LIN {X -76.668,Y -27.149,Z -45.520,A -90.000,B 90.000,C 0.000} C_DIS
LIN {X -76.579,Y -27.148,Z -45.468,A -90.000,B 90.000,C 0.000} C_DIS
LIN {X -76.520,Y -27.146,Z -45.437,A -90.000,B 90.000,C 0.000} C_DIS
LIN {X -76.472,Y -27.145,Z -45.413,A -90.000,B 90.000,C 0.000} C_DIS
LIN {X -76.330,Y -27.139,Z -45.352,A -90.000,B 90.000,C 0.000} C_DIS
LIN {X -76.220,Y -27.135,Z -45.309,A -90.000,B 90.000,C 0.000} C_DIS
LIN {X -75.832,Y -27.123,Z -45.175,A -90.000,B 90.000,C 0.000} C_DIS
LIN {X -75.654,Y -27.113,Z -45.115,A -90.000,B 90.000,C 0.000} C_DIS
LIN {X -75.440,Y -27.095,Z -45.043,A -90.000,B 90.000,C 0.000} C_DIS
LIN {X -75.320,Y -27.086,Z -45.007,A -90.000,B 90.000,C 0.000} C_DIS
LIN {X -75.000,Y -27.064,Z -44.932,A -90.000,B 90.000,C 0.000} C_DIS
LIN {X -74.933,Y -27.060,Z -44.917,A -90.000,B 90.000,C 0.000} C_DIS
LIN {X -74.743,Y -27.049,Z -44.886,A -90.000,B 90.000,C 0.000} C_DIS
LIN {X -74.638,Y -27.044,Z -44.876,A -90.000,B 90.000,C 0.000} C_DIS
LIN {X -74.553,Y -27.040,Z -44.872,A -90.000,B 90.000,C 0.000} C_DIS
LIN {X -74.405,Y -27.038,Z -44.874,A -90.000,B 90.000,C 0.000} C_DIS
LIN {X -74.238,Y -27.035,Z -44.881,A -90.000,B 90.000,C 0.000} C_DIS
LIN {X -74.171,Y -27.032,Z -44.885,A -90.000,B 90.000,C 0.000} C_DIS
LIN {X -74.041,Y -27.028,Z -44.899,A -90.000,B 90.000,C 0.000} C_DIS
LIN {X -73.894,Y -27.024,Z -44.925,A -90.000,B 90.000,C 0.000} C_DIS
LIN {X -73.078,Y -26.996,Z -45.023,A -90.000,B 90.000,C 0.000} C_DIS
LIN {X -72.681,Y -26.986,Z -45.070,A -90.000,B 90.000,C 0.000} C_DIS
LIN {X -72.606,Y -26.984,Z -45.081,A -90.000,B 90.000,C 0.000} C_DIS
LIN {X -72.312,Y -26.976,Z -45.155,A -90.000,B 90.000,C 0.000} C_DIS
LIN {X -72.076,Y -26.973,Z -45.234,A -90.000,B 90.000,C 0.000} C_DIS
LIN {X -72.048,Y -26.973,Z -45.245,A -90.000,B 90.000,C 0.000} C_DIS
LIN {X -71.550,Y -26.959,Z -45.362,A -90.000,B 90.000,C 0.000} C_DIS
LIN {X -71.035,Y -26.949,Z -45.481,A -90.000,B 90.000,C 0.000} C_DIS
LIN {X -70.942,Y -26.945,Z -45.503,A -90.000,B 90.000,C 0.000} C_DIS
LIN {X -70.816,Y -26.940,Z -45.537,A -90.000,B 90.000,C 0.000} C_DIS
LIN {X -70.607,Y -26.935,Z -45.607,A -90.000,B 90.000,C 0.000} C_DIS
LIN {X -70.486,Y -26.933,Z -45.651,A -90.000,B 90.000,C 0.000} C_DIS
LIN {X -69.761,Y -26.903,Z -45.823,A -90.000,B 90.000,C 0.000} C_DIS
LIN {X -69.366,Y -26.892,Z -45.916,A -90.000,B 90.000,C 0.000} C_DIS
LIN {X -69.227,Y -26.882,Z -45.922,A -90.000,B 90.000,C 0.000} C_DIS
LIN {X -69.048,Y -26.872,Z -45.944,A -90.000,B 90.000,C 0.000} C_DIS
LIN {X -68.707,Y -26.860,Z -46.014,A -90.000,B 90.000,C 0.000} C_DIS
LIN {X -67.594,Y -26.796,Z -46.253,A -90.000,B 90.000,C 0.000} C_DIS
LIN {X -67.151,Y -26.765,Z -46.342,A -90.000,B 90.000,C 0.000} C_DIS
LIN {X -66.963,Y -26.753,Z -46.384,A -90.000,B 90.000,C 0.000} C_DIS
LIN {X -66.920,Y -26.749,Z -46.390,A -90.000,B 90.000,C 0.000} C_DIS
LIN {X -66.399,Y -26.719,Z -46.458,A -90.000,B 90.000,C 0.000} C_DIS
LIN {X -66.250,Y -26.713,Z -46.485,A -90.000,B 90.000,C 0.000} C_DIS
LIN {X -66.013,Y -26.705,Z -46.537,A -90.000,B 90.000,C 0.000} C_DIS
LIN {X -65.089,Y -26.644,Z -46.751,A -90.000,B 90.000,C 0.000} C_DIS
LIN {X -64.621,Y -26.614,Z -46.860,A -90.000,B 90.000,C 0.000} C_DIS
LIN {X -64.516,Y -26.603,Z -46.873,A -90.000,B 90.000,C 0.000} C_DIS
LIN {X -64.385,Y -26.595,Z -46.892,A -90.000,B 90.000,C 0.000} C_DIS
LIN {X -64.154,Y -26.585,Z -46.933,A -90.000,B 90.000,C 0.000} C_DIS
LIN {X -63.476,Y -26.545,Z -47.056,A -90.000,B 90.000,C 0.000} C_DIS
LIN {X -63.310,Y -26.538,Z -47.093,A -90.000,B 90.000,C 0.000} C_DIS
LIN {X -63.159,Y -26.532,Z -47.128,A -90.000,B 90.000,C 0.000} C_DIS
LIN {X -61.858,Y -26.456,Z -47.450,A -90.000,B 90.000,C 0.000} C_DIS
LIN {X -61.801,Y -26.451,Z -47.460,A -90.000,B 90.000,C 0.000} C_DIS
LIN {X -61.487,Y -26.434,Z -47.509,A -90.000,B 90.000,C 0.000} C_DIS
LIN {X -61.371,Y -26.430,Z -47.531,A -90.000,B 90.000,C 0.000} C_DIS
LIN {X -61.170,Y -26.422,Z -47.574,A -90.000,B 90.000,C 0.000} C_DIS
LIN {X -60.377,Y -26.379,Z -47.754,A -90.000,B 90.000,C 0.000} C_DIS
LIN {X -59.277,Y -26.330,Z -48.032,A -90.000,B 90.000,C 0.000} C_DIS
LIN {X -59.103,Y -26.323,Z -48.077,A -90.000,B 90.000,C 0.000} C_DIS
LIN {X -59.005,Y -26.321,Z -48.100,A -90.000,B 90.000,C 0.000} C_DIS
LIN {X -58.397,Y -26.301,Z -48.215,A -90.000,B 90.000,C 0.000} C_DIS
LIN {X -58.186,Y -26.296,Z -48.262,A -90.000,B 90.000,C 0.000} C_DIS
LIN {X -57.425,Y -26.286,Z -48.443,A -90.000,B 90.000,C 0.000} C_DIS
LIN {X -56.485,Y -26.265,Z -48.675,A -90.000,B 90.000,C 0.000} C_DIS
LIN {X -55.979,Y -26.267,Z -48.792,A -90.000,B 90.000,C 0.000} C_DIS
LIN {X -55.691,Y -26.263,Z -48.851,A -90.000,B 90.000,C 0.000} C_DIS
LIN {X -54.901,Y -26.262,Z -49.008,A -90.000,B 90.000,C 0.000} C_DIS
LIN {X -54.076,Y -26.270,Z -49.199,A -90.000,B 90.000,C 0.000} C_DIS
LIN {X -52.954,Y -26.306,Z -49.443,A -90.000,B 90.000,C 0.000} C_DIS
LIN {X -51.548,Y -26.347,Z -49.740,A -90.000,B 90.000,C 0.000} C_DIS
LIN {X -51.220,Y -26.356,Z -49.809,A -90.000,B 90.000,C 0.000} C_DIS
LIN {X -50.961,Y -26.369,Z -49.862,A -90.000,B 90.000,C 0.000} C_DIS
LIN {X -50.773,Y -26.379,Z -49.904,A -90.000,B 90.000,C 0.000} C_DIS
LIN {X -50.032,Y -26.422,Z -50.072,A -90.000,B 90.000,C 0.000} C_DIS
LIN {X -49.104,Y -26.464,Z -50.267,A -90.000,B 90.000,C 0.000} C_DIS
LIN {X -48.814,Y -26.479,Z -50.333,A -90.000,B 90.000,C 0.000} C_DIS
LIN {X -48.233,Y -26.506,Z -50.468,A -90.000,B 90.000,C 0.000} C_DIS
LIN {X -47.893,Y -26.526,Z -50.543,A -90.000,B 90.000,C 0.000} C_DIS
LIN {X -47.412,Y -26.550,Z -50.637,A -90.000,B 90.000,C 0.000} C_DIS
LIN {X -46.971,Y -26.573,Z -50.730,A -90.000,B 90.000,C 0.000} C_DIS
LIN {X -46.694,Y -26.575,Z -50.762,A -90.000,B 90.000,C 0.000} C_DIS
LIN {X -45.976,Y -26.553,Z -50.795,A -90.000,B 90.000,C 0.000} C_DIS
LIN {X -45.116,Y -26.531,Z -50.839,A -90.000,B 90.000,C 0.000} C_DIS
LIN {X -44.321,Y -26.510,Z -50.871,A -90.000,B 90.000,C 0.000} C_DIS
LIN {X -43.871,Y -26.485,Z -50.896,A -90.000,B 90.000,C 0.000} C_DIS
LIN {X -42.715,Y -26.432,Z -50.983,A -90.000,B 90.000,C 0.000} C_DIS
LIN {X -42.367,Y -26.419,Z -51.020,A -90.000,B 90.000,C 0.000} C_DIS
LIN {X -41.622,Y -26.397,Z -51.105,A -90.000,B 90.000,C 0.000} C_DIS
LIN {X -40.921,Y -26.380,Z -51.187,A -90.000,B 90.000,C 0.000} C_DIS
LIN {X -39.390,Y -26.335,Z -51.371,A -90.000,B 90.000,C 0.000} C_DIS
LIN {X -39.171,Y -26.331,Z -51.405,A -90.000,B 90.000,C 0.000} C_DIS
LIN {X -38.129,Y -26.312,Z -51.576,A -90.000,B 90.000,C 0.000} C_DIS
LIN {X -37.797,Y -26.306,Z -51.632,A -90.000,B 90.000,C 0.000} C_DIS
LIN {X -37.029,Y -26.296,Z -51.768,A -90.000,B 90.000,C 0.000} C_DIS
LIN {X -36.278,Y -26.283,Z -51.903,A -90.000,B 90.000,C 0.000} C_DIS
LIN {X -35.844,Y -26.277,Z -51.985,A -90.000,B 90.000,C 0.000} C_DIS
LIN {X -35.325,Y -26.267,Z -52.085,A -90.000,B 90.000,C 0.000} C_DIS
LIN {X -33.082,Y -26.239,Z -52.548,A -90.000,B 90.000,C 0.000} C_DIS
LIN {X -32.307,Y -26.223,Z -52.710,A -90.000,B 90.000,C 0.000} C_DIS
LIN {X -31.608,Y -26.212,Z -52.862,A -90.000,B 90.000,C 0.000} C_DIS
LIN {X -30.365,Y -26.201,Z -53.148,A -90.000,B 90.000,C 0.000} C_DIS
LIN {X -29.820,Y -26.194,Z -53.275,A -90.000,B 90.000,C 0.000} C_DIS
LIN {X -29.558,Y -26.188,Z -53.337,A -90.000,B 90.000,C 0.000} C_DIS
LIN {X -29.212,Y -26.184,Z -53.417,A -90.000,B 90.000,C 0.000} C_DIS
LIN {X -27.279,Y -26.151,Z -53.851,A -90.000,B 90.000,C 0.000} C_DIS
LIN {X -26.462,Y -26.136,Z -54.036,A -90.000,B 90.000,C 0.000} C_DIS
LIN {X -26.354,Y -26.132,Z -54.059,A -90.000,B 90.000,C 0.000} C_DIS
LIN {X -24.983,Y -26.105,Z -54.333,A -90.000,B 90.000,C 0.000} C_DIS
LIN {X -24.301,Y -26.086,Z -54.456,A -90.000,B 90.000,C 0.000} C_DIS
LIN {X -23.848,Y -26.066,Z -54.528,A -90.000,B 90.000,C 0.000} C_DIS
LIN {X -23.603,Y -26.060,Z -54.564,A -90.000,B 90.000,C 0.000} C_DIS
LIN {X -23.357,Y -26.057,Z -54.597,A -90.000,B 90.000,C 0.000} C_DIS
LIN {X -22.651,Y -26.032,Z -54.669,A -90.000,B 90.000,C 0.000} C_DIS
LIN {X -22.402,Y -26.017,Z -54.685,A -90.000,B 90.000,C 0.000} C_DIS
LIN {X -22.145,Y -25.999,Z -54.688,A -90.000,B 90.000,C 0.000} C_DIS
LIN {X -21.779,Y -25.983,Z -54.683,A -90.000,B 90.000,C 0.000} C_DIS
LIN {X -21.198,Y -25.921,Z -54.631,A -90.000,B 90.000,C 0.000} C_DIS
LIN {X -21.158,Y -25.919,Z -54.625,A -90.000,B 90.000,C 0.000} C_DIS
LIN {X -20.482,Y -25.823,Z -54.462,A -90.000,B 90.000,C 0.000} C_DIS
LIN {X -20.459,Y -25.820,Z -54.457,A -90.000,B 90.000,C 0.000} C_DIS
LIN {X -20.316,Y -25.816,Z -54.414,A -90.000,B 90.000,C 0.000} C_DIS
LIN {X -19.976,Y -25.803,Z -54.320,A -90.000,B 90.000,C 0.000} C_DIS
LIN {X -19.491,Y -25.762,Z -54.163,A -90.000,B 90.000,C 0.000} C_DIS
LIN {X -19.170,Y -25.749,Z -54.042,A -90.000,B 90.000,C 0.000} C_DIS
LIN {X -18.511,Y -25.729,Z -53.805,A -90.000,B 90.000,C 0.000} C_DIS
LIN {X -18.354,Y -25.723,Z -53.745,A -90.000,B 90.000,C 0.000} C_DIS
LIN {X -17.302,Y -25.718,Z -53.351,A -90.000,B 90.000,C 0.000} C_DIS
LIN {X -16.990,Y -25.716,Z -53.234,A -90.000,B 90.000,C 0.000} C_DIS
LIN {X -16.551,Y -25.702,Z -53.087,A -90.000,B 90.000,C 0.000} C_DIS
LIN {X -16.275,Y -25.697,Z -52.992,A -90.000,B 90.000,C 0.000} C_DIS
LIN {X -15.804,Y -25.701,Z -52.842,A -90.000,B 90.000,C 0.000} C_DIS
LIN {X -15.519,Y -25.709,Z -52.757,A -90.000,B 90.000,C 0.000} C_DIS
LIN {X -14.893,Y -25.715,Z -52.585,A -90.000,B 90.000,C 0.000} C_DIS
LIN {X -14.842,Y -25.713,Z -52.574,A -90.000,B 90.000,C 0.000} C_DIS
LIN {X -14.139,Y -25.698,Z -52.428,A -90.000,B 90.000,C 0.000} C_DIS
LIN {X -13.133,Y -25.670,Z -52.234,A -90.000,B 90.000,C 0.000} C_DIS
LIN {X -12.867,Y -25.665,Z -52.190,A -90.000,B 90.000,C 0.000} C_DIS
LIN {X -12.574,Y -25.660,Z -52.144,A -90.000,B 90.000,C 0.000} C_DIS
LIN {X -11.885,Y -25.673,Z -52.058,A -90.000,B 90.000,C 0.000} C_DIS
LIN {X -11.634,Y -25.672,Z -52.037,A -90.000,B 90.000,C 0.000} C_DIS
LIN {X -11.198,Y -25.673,Z -52.007,A -90.000,B 90.000,C 0.000} C_DIS
LIN {X -10.131,Y -25.674,Z -51.968,A -90.000,B 90.000,C 0.000} C_DIS
LIN {X -9.127,Y -25.674,Z -51.924,A -90.000,B 90.000,C 0.000} C_DIS
LIN {X -9.054,Y -25.675,Z -51.922,A -90.000,B 90.000,C 0.000} C_DIS
LIN {X -8.312,Y -25.671,Z -51.917,A -90.000,B 90.000,C 0.000} C_DIS
LIN {X -7.938,Y -25.680,Z -51.922,A -90.000,B 90.000,C 0.000} C_DIS
LIN {X -7.084,Y -25.713,Z -51.944,A -90.000,B 90.000,C 0.000} C_DIS
LIN {X -6.515,Y -25.723,Z -51.975,A -90.000,B 90.000,C 0.000} C_DIS
LIN {X -5.811,Y -25.734,Z -52.016,A -90.000,B 90.000,C 0.000} C_DIS
LIN {X -5.328,Y -25.747,Z -52.047,A -90.000,B 90.000,C 0.000} C_DIS
LIN {X -4.775,Y -25.774,Z -52.093,A -90.000,B 90.000,C 0.000} C_DIS
LIN {X -3.453,Y -25.814,Z -52.238,A -90.000,B 90.000,C 0.000} C_DIS
LIN {X -2.718,Y -25.836,Z -52.319,A -90.000,B 90.000,C 0.000} C_DIS
LIN {X -2.230,Y -25.852,Z -52.374,A -90.000,B 90.000,C 0.000} C_DIS
LIN {X -1.872,Y -25.876,Z -52.429,A -90.000,B 90.000,C 0.000} C_DIS
LIN {X -0.557,Y -25.960,Z -52.642,A -90.000,B 90.000,C 0.000} C_DIS
LIN {X -0.166,Y -25.976,Z -52.698,A -90.000,B 90.000,C 0.000} C_DIS
LIN {X 0.552,Y -26.009,Z -52.808,A -90.000,B 90.000,C 0.000} C_DIS
LIN {X 0.727,Y -26.014,Z -52.838,A -90.000,B 90.000,C 0.000} C_DIS
LIN {X 0.921,Y -26.024,Z -52.878,A -90.000,B 90.000,C 0.000} C_DIS
LIN {X 1.351,Y -26.042,Z -52.975,A -90.000,B 90.000,C 0.000} C_DIS
LIN {X 1.495,Y -26.054,Z -53.002,A -90.000,B 90.000,C 0.000} C_DIS
LIN {X 2.799,Y -26.132,Z -53.211,A -90.000,B 90.000,C 0.000} C_DIS
LIN {X 3.009,Y -26.149,Z -53.251,A -90.000,B 90.000,C 0.000} C_DIS
LIN {X 3.118,Y -26.159,Z -53.272,A -90.000,B 90.000,C 0.000} C_DIS
LIN {X 3.768,Y -26.195,Z -53.373,A -90.000,B 90.000,C 0.000} C_DIS
LIN {X 4.343,Y -26.230,Z -53.460,A -90.000,B 90.000,C 0.000} C_DIS
LIN {X 4.515,Y -26.234,Z -53.477,A -90.000,B 90.000,C 0.000} C_DIS
LIN {X 4.986,Y -26.259,Z -53.514,A -90.000,B 90.000,C 0.000} C_DIS
LIN {X 5.416,Y -26.287,Z -53.555,A -90.000,B 90.000,C 0.000} C_DIS
LIN {X 5.715,Y -26.295,Z -53.563,A -90.000,B 90.000,C 0.000} C_DIS
LIN {X 6.310,Y -26.301,Z -53.557,A -90.000,B 90.000,C 0.000} C_DIS
LIN {X 6.763,Y -26.310,Z -53.550,A -90.000,B 90.000,C 0.000} C_DIS
LIN {X 7.708,Y -26.306,Z -53.477,A -90.000,B 90.000,C 0.000} C_DIS
LIN {X 8.237,Y -26.294,Z -53.427,A -90.000,B 90.000,C 0.000} C_DIS
LIN {X 8.504,Y -26.288,Z -53.400,A -90.000,B 90.000,C 0.000} C_DIS
LIN {X 9.112,Y -26.249,Z -53.356,A -90.000,B 90.000,C 0.000} C_DIS
LIN {X 9.378,Y -26.233,Z -53.345,A -90.000,B 90.000,C 0.000} C_DIS
LIN {X 9.815,Y -26.206,Z -53.332,A -90.000,B 90.000,C 0.000} C_DIS
LIN {X 9.935,Y -26.202,Z -53.332,A -90.000,B 90.000,C 0.000} C_DIS
LIN {X 10.931,Y -26.179,Z -53.355,A -90.000,B 90.000,C 0.000} C_DIS
LIN {X 11.248,Y -26.159,Z -53.373,A -90.000,B 90.000,C 0.000} C_DIS
LIN {X 11.681,Y -26.144,Z -53.417,A -90.000,B 90.000,C 0.000} C_DIS
LIN {X 11.767,Y -26.143,Z -53.430,A -90.000,B 90.000,C 0.000} C_DIS
LIN {X 12.047,Y -26.130,Z -53.483,A -90.000,B 90.000,C 0.000} C_DIS
LIN {X 12.477,Y -26.118,Z -53.558,A -90.000,B 90.000,C 0.000} C_DIS
LIN {X 12.961,Y -26.073,Z -53.618,A -90.000,B 90.000,C 0.000} C_DIS
LIN {X 13.125,Y -26.063,Z -53.643,A -90.000,B 90.000,C 0.000} C_DIS
LIN {X 13.751,Y -26.044,Z -53.760,A -90.000,B 90.000,C 0.000} C_DIS
LIN {X 14.266,Y -26.019,Z -53.825,A -90.000,B 90.000,C 0.000} C_DIS
LIN {X 14.500,Y -26.013,Z -53.861,A -90.000,B 90.000,C 0.000} C_DIS
LIN {X 14.939,Y -26.001,Z -53.932,A -90.000,B 90.000,C 0.000} C_DIS
LIN {X 15.047,Y -25.993,Z -53.945,A -90.000,B 90.000,C 0.000} C_DIS
LIN {X 15.382,Y -25.981,Z -53.980,A -90.000,B 90.000,C 0.000} C_DIS
LIN {X 15.560,Y -25.978,Z -54.003,A -90.000,B 90.000,C 0.000} C_DIS
LIN {X 15.976,Y -25.953,Z -54.039,A -90.000,B 90.000,C 0.000} C_DIS
LIN {X 16.371,Y -25.945,Z -54.086,A -90.000,B 90.000,C 0.000} C_DIS
LIN {X 16.524,Y -25.935,Z -54.097,A -90.000,B 90.000,C 0.000} C_DIS
LIN {X 16.741,Y -26.026,Z -54.021,A -90.000,B 90.000,C 0.000} C_DIS
LIN {X 16.808,Y -26.055,Z -54.000,A -90.000,B 90.000,C 0.000} C_DIS
LIN {X 16.933,Y -26.108,Z -53.971,A -90.000,B 90.000,C 0.000} C_DIS
LIN {X 17.083,Y -26.172,Z -53.944,A -90.000,B 90.000,C 0.000} C_DIS
LIN {X 17.196,Y -26.216,Z -53.927,A -90.000,B 90.000,C 0.000} C_DIS
LIN {X 17.303,Y -26.254,Z -53.911,A -90.000,B 90.000,C 0.000} C_DIS
LIN {X 17.592,Y -26.359,Z -53.877,A -90.000,B 90.000,C 0.000} C_DIS
LIN {X 17.749,Y -26.413,Z -53.864,A -90.000,B 90.000,C 0.000} C_DIS
LIN {X 17.828,Y -26.441,Z -53.862,A -90.000,B 90.000,C 0.000} C_DIS
LIN {X 18.139,Y -26.545,Z -53.863,A -90.000,B 90.000,C 0.000} C_DIS
LIN {X 18.300,Y -26.602,Z -53.870,A -90.000,B 90.000,C 0.000} C_DIS
LIN {X 18.401,Y -26.638,Z -53.867,A -90.000,B 90.000,C 0.000} C_DIS
LIN {X 18.613,Y -26.714,Z -53.875,A -90.000,B 90.000,C 0.000} C_DIS
LIN {X 18.655,Y -26.729,Z -53.880,A -90.000,B 90.000,C 0.000} C_DIS
LIN {X 18.754,Y -26.750,Z -53.795,A -90.000,B 90.000,C 0.000} C_DIS
LIN {X 18.774,Y -26.736,Z -53.643,A -90.000,B 90.000,C 0.000} C_DIS
LIN {X 18.828,Y -26.717,Z -53.412,A -90.000,B 90.000,C 0.000} C_DIS
LIN {X 18.955,Y -26.695,Z -53.020,A -90.000,B 90.000,C 0.000} C_DIS
LIN {X 19.026,Y -26.673,Z -52.812,A -90.000,B 90.000,C 0.000} C_DIS
LIN {X 19.080,Y -26.660,Z -52.672,A -90.000,B 90.000,C 0.000} C_DIS
LIN {X 19.259,Y -26.627,Z -52.252,A -90.000,B 90.000,C 0.000} C_DIS
LIN {X 19.331,Y -26.607,Z -52.091,A -90.000,B 90.000,C 0.000} C_DIS
LIN {X 19.446,Y -26.577,Z -51.845,A -90.000,B 90.000,C 0.000} C_DIS
LIN {X 19.492,Y -26.567,Z -51.753,A -90.000,B 90.000,C 0.000} C_DIS
LIN {X 19.554,Y -26.558,Z -51.644,A -90.000,B 90.000,C 0.000} C_DIS
LIN {X 19.612,Y -26.551,Z -51.554,A -90.000,B 90.000,C 0.000} C_DIS
LIN {X 19.696,Y -26.542,Z -51.430,A -90.000,B 90.000,C 0.000} C_DIS
LIN {X 19.880,Y -26.514,Z -51.172,A -90.000,B 90.000,C 0.000} C_DIS
LIN {X 20.028,Y -26.490,Z -50.967,A -90.000,B 90.000,C 0.000} C_DIS
LIN {X 20.210,Y -26.458,Z -50.712,A -90.000,B 90.000,C 0.000} C_DIS
LIN {X 20.290,Y -26.447,Z -50.610,A -90.000,B 90.000,C 0.000} C_DIS
LIN {X 20.384,Y -26.435,Z -50.495,A -90.000,B 90.000,C 0.000} C_DIS
LIN {X 20.492,Y -26.416,Z -50.351,A -90.000,B 90.000,C 0.000} C_DIS
LIN {X 20.559,Y -26.405,Z -50.264,A -90.000,B 90.000,C 0.000} C_DIS
LIN {X 20.692,Y -26.388,Z -50.109,A -90.000,B 90.000,C 0.000} C_DIS
LIN {X 20.911,Y -26.361,Z -49.879,A -90.000,B 90.000,C 0.000} C_DIS
LIN {X 21.128,Y -26.327,Z -49.657,A -90.000,B 90.000,C 0.000} C_DIS
LIN {X 21.369,Y -26.295,Z -49.419,A -90.000,B 90.000,C 0.000} C_DIS
LIN {X 21.491,Y -26.280,Z -49.298,A -90.000,B 90.000,C 0.000} C_DIS
LIN {X 21.593,Y -26.271,Z -49.204,A -90.000,B 90.000,C 0.000} C_DIS
LIN {X 21.776,Y -26.243,Z -49.013,A -90.000,B 90.000,C 0.000} C_DIS
LIN {X 21.928,Y -26.228,Z -48.873,A -90.000,B 90.000,C 0.000} C_DIS
LIN {X 22.146,Y -26.201,Z -48.678,A -90.000,B 90.000,C 0.000} C_DIS
LIN {X 22.398,Y -26.169,Z -48.453,A -90.000,B 90.000,C 0.000} C_DIS
LIN {X 22.719,Y -26.122,Z -48.184,A -90.000,B 90.000,C 0.000} C_DIS
LIN {X 22.870,Y -26.096,Z -48.043,A -90.000,B 90.000,C 0.000} C_DIS
LIN {X 23.304,Y -26.044,Z -47.683,A -90.000,B 90.000,C 0.000} C_DIS
LIN {X 23.430,Y -26.028,Z -47.580,A -90.000,B 90.000,C 0.000} C_DIS
LIN {X 23.577,Y -26.006,Z -47.467,A -90.000,B 90.000,C 0.000} C_DIS
LIN {X 23.702,Y -25.988,Z -47.374,A -90.000,B 90.000,C 0.000} C_DIS
LIN {X 23.939,Y -25.949,Z -47.209,A -90.000,B 90.000,C 0.000} C_DIS
LIN {X 23.988,Y -25.939,Z -47.172,A -90.000,B 90.000,C 0.000} C_DIS
LIN {X 24.179,Y -25.908,Z -47.041,A -90.000,B 90.000,C 0.000} C_DIS
LIN {X 24.532,Y -25.864,Z -46.789,A -90.000,B 90.000,C 0.000} C_DIS
LIN {X 24.820,Y -25.823,Z -46.595,A -90.000,B 90.000,C 0.000} C_DIS
LIN {X 25.032,Y -25.794,Z -46.461,A -90.000,B 90.000,C 0.000} C_DIS
LIN {X 25.512,Y -25.738,Z -46.177,A -90.000,B 90.000,C 0.000} C_DIS
LIN {X 25.704,Y -25.713,Z -46.074,A -90.000,B 90.000,C 0.000} C_DIS
LIN {X 25.770,Y -25.706,Z -46.039,A -90.000,B 90.000,C 0.000} C_DIS
LIN {X 25.938,Y -25.679,Z -45.945,A -90.000,B 90.000,C 0.000} C_DIS
LIN {X 25.999,Y -25.672,Z -45.913,A -90.000,B 90.000,C 0.000} C_DIS
LIN {X 26.061,Y -25.662,Z -45.884,A -90.000,B 90.000,C 0.000} C_DIS
LIN {X 26.279,Y -25.639,Z -45.764,A -90.000,B 90.000,C 0.000} C_DIS
LIN {X 26.350,Y -25.630,Z -45.729,A -90.000,B 90.000,C 0.000} C_DIS
LIN {X 26.679,Y -25.600,Z -45.574,A -90.000,B 90.000,C 0.000} C_DIS
LIN {X 26.829,Y -25.586,Z -45.504,A -90.000,B 90.000,C 0.000} C_DIS
LIN {X 27.144,Y -25.554,Z -45.370,A -90.000,B 90.000,C 0.000} C_DIS
LIN {X 27.283,Y -25.545,Z -45.313,A -90.000,B 90.000,C 0.000} C_DIS
LIN {X 27.612,Y -25.519,Z -45.199,A -90.000,B 90.000,C 0.000} C_DIS
LIN {X 27.822,Y -25.503,Z -45.125,A -90.000,B 90.000,C 0.000} C_DIS
LIN {X 28.017,Y -25.494,Z -45.048,A -90.000,B 90.000,C 0.000} C_DIS
LIN {X 28.430,Y -25.472,Z -44.901,A -90.000,B 90.000,C 0.000} C_DIS
LIN {X 28.884,Y -25.440,Z -44.766,A -90.000,B 90.000,C 0.000} C_DIS
LIN {X 29.328,Y -25.418,Z -44.640,A -90.000,B 90.000,C 0.000} C_DIS
LIN {X 29.665,Y -25.409,Z -44.546,A -90.000,B 90.000,C 0.000} C_DIS
LIN {X 30.143,Y -25.387,Z -44.458,A -90.000,B 90.000,C 0.000} C_DIS
LIN {X 30.385,Y -25.381,Z -44.414,A -90.000,B 90.000,C 0.000} C_DIS
LIN {X 30.701,Y -25.375,Z -44.351,A -90.000,B 90.000,C 0.000} C_DIS
LIN {X 30.921,Y -25.375,Z -44.308,A -90.000,B 90.000,C 0.000} C_DIS
LIN {X 31.396,Y -25.369,Z -44.241,A -90.000,B 90.000,C 0.000} C_DIS
LIN {X 31.533,Y -25.366,Z -44.225,A -90.000,B 90.000,C 0.000} C_DIS
LIN {X 31.992,Y -25.366,Z -44.150,A -90.000,B 90.000,C 0.000} C_DIS
LIN {X 32.576,Y -25.362,Z -44.091,A -90.000,B 90.000,C 0.000} C_DIS
LIN {X 32.639,Y -25.362,Z -44.084,A -90.000,B 90.000,C 0.000} C_DIS
LIN {X 33.254,Y -25.365,Z -44.001,A -90.000,B 90.000,C 0.000} C_DIS
LIN {X 33.639,Y -25.384,Z -43.913,A -90.000,B 90.000,C 0.000} C_DIS
LIN {X 34.121,Y -25.420,Z -43.779,A -90.000,B 90.000,C 0.000} C_DIS
LIN {X 34.426,Y -25.447,Z -43.697,A -90.000,B 90.000,C 0.000} C_DIS
LIN {X 34.840,Y -25.491,Z -43.589,A -90.000,B 90.000,C 0.000} C_DIS
LIN {X 35.180,Y -25.532,Z -43.503,A -90.000,B 90.000,C 0.000} C_DIS
LIN {X 35.643,Y -25.595,Z -43.382,A -90.000,B 90.000,C 0.000} C_DIS
LIN {X 35.904,Y -25.637,Z -43.319,A -90.000,B 90.000,C 0.000} C_DIS
LIN {X 36.220,Y -25.677,Z -43.233,A -90.000,B 90.000,C 0.000} C_DIS
LIN {X 36.547,Y -25.697,Z -43.128,A -90.000,B 90.000,C 0.000} C_DIS
LIN {X 37.209,Y -25.708,Z -42.887,A -90.000,B 90.000,C 0.000} C_DIS
LIN {X 37.591,Y -25.709,Z -42.757,A -90.000,B 90.000,C 0.000} C_DIS
LIN {X 38.265,Y -25.703,Z -42.524,A -90.000,B 90.000,C 0.000} C_DIS
LIN {X 39.037,Y -25.689,Z -42.263,A -90.000,B 90.000,C 0.000} C_DIS
LIN {X 39.260,Y -25.683,Z -42.190,A -90.000,B 90.000,C 0.000} C_DIS
LIN {X 39.448,Y -25.682,Z -42.131,A -90.000,B 90.000,C 0.000} C_DIS
LIN {X 40.472,Y -25.649,Z -41.869,A -90.000,B 90.000,C 0.000} C_DIS
LIN {X 40.807,Y -25.638,Z -41.786,A -90.000,B 90.000,C 0.000} C_DIS
LIN {X 40.945,Y -25.635,Z -41.753,A -90.000,B 90.000,C 0.000} C_DIS
LIN {X 41.621,Y -25.601,Z -41.626,A -90.000,B 90.000,C 0.000} C_DIS
LIN {X 42.277,Y -25.590,Z -41.517,A -90.000,B 90.000,C 0.000} C_DIS
LIN {X 42.441,Y -25.586,Z -41.493,A -90.000,B 90.000,C 0.000} C_DIS
LIN {X 42.768,Y -25.584,Z -41.450,A -90.000,B 90.000,C 0.000} C_DIS
LIN {X 42.836,Y -25.581,Z -41.444,A -90.000,B 90.000,C 0.000} C_DIS
LIN {X 43.470,Y -25.549,Z -41.413,A -90.000,B 90.000,C 0.000} C_DIS
LIN {X 43.740,Y -25.536,Z -41.407,A -90.000,B 90.000,C 0.000} C_DIS
LIN {X 44.495,Y -25.521,Z -41.402,A -90.000,B 90.000,C 0.000} C_DIS
LIN {X 44.954,Y -25.510,Z -41.405,A -90.000,B 90.000,C 0.000} C_DIS
LIN {X 45.185,Y -25.496,Z -41.424,A -90.000,B 90.000,C 0.000} C_DIS
LIN {X 45.672,Y -25.474,Z -41.464,A -90.000,B 90.000,C 0.000} C_DIS
LIN {X 45.840,Y -25.472,Z -41.480,A -90.000,B 90.000,C 0.000} C_DIS
LIN {X 46.338,Y -25.470,Z -41.531,A -90.000,B 90.000,C 0.000} C_DIS
LIN {X 46.541,Y -25.470,Z -41.554,A -90.000,B 90.000,C 0.000} C_DIS
LIN {X 46.945,Y -25.470,Z -41.607,A -90.000,B 90.000,C 0.000} C_DIS
LIN {X 46.969,Y -25.470,Z -41.610,A -90.000,B 90.000,C 0.000} C_DIS
LIN {X 47.006,Y -25.470,Z -41.616,A -90.000,B 90.000,C 0.000} C_DIS
LIN {X 47.631,Y -25.452,Z -41.759,A -90.000,B 90.000,C 0.000} C_DIS
LIN {X 48.069,Y -25.437,Z -41.870,A -90.000,B 90.000,C 0.000} C_DIS
LIN {X 49.214,Y -25.419,Z -42.200,A -90.000,B 90.000,C 0.000} C_DIS
LIN {X 49.936,Y -25.396,Z -42.449,A -90.000,B 90.000,C 0.000} C_DIS
LIN {X 50.448,Y -25.395,Z -42.631,A -90.000,B 90.000,C 0.000} C_DIS
LIN {X 50.890,Y -25.395,Z -42.799,A -90.000,B 90.000,C 0.000} C_DIS
LIN {X 51.270,Y -25.390,Z -42.968,A -90.000,B 90.000,C 0.000} C_DIS
LIN {X 51.726,Y -25.382,Z -43.186,A -90.000,B 90.000,C 0.000} C_DIS
LIN {X 52.514,Y -25.375,Z -43.567,A -90.000,B 90.000,C 0.000} C_DIS
LIN {X 52.832,Y -25.375,Z -43.721,A -90.000,B 90.000,C 0.000} C_DIS
LIN {X 53.252,Y -25.371,Z -43.942,A -90.000,B 90.000,C 0.000} C_DIS
LIN {X 53.731,Y -25.369,Z -44.197,A -90.000,B 90.000,C 0.000} C_DIS
LIN {X 54.062,Y -25.373,Z -44.381,A -90.000,B 90.000,C 0.000} C_DIS
LIN {X 54.663,Y -25.366,Z -44.782,A -90.000,B 90.000,C 0.000} C_DIS
LIN {X 55.983,Y -25.353,Z -45.672,A -90.000,B 90.000,C 0.000} C_DIS
LIN {X 56.709,Y -25.348,Z -46.165,A -90.000,B 90.000,C 0.000} C_DIS
LIN {X 56.970,Y -25.353,Z -46.344,A -90.000,B 90.000,C 0.000} C_DIS
LIN {X 57.628,Y -25.350,Z -46.890,A -90.000,B 90.000,C 0.000} C_DIS
LIN {X 58.716,Y -25.347,Z -47.797,A -90.000,B 90.000,C 0.000} C_DIS
LIN {X 59.365,Y -25.346,Z -48.341,A -90.000,B 90.000,C 0.000} C_DIS
LIN {X 59.550,Y -25.348,Z -48.500,A -90.000,B 90.000,C 0.000} C_DIS
LIN {X 61.659,Y -25.345,Z -50.511,A -90.000,B 90.000,C 0.000} C_DIS
LIN {X 62.243,Y -25.345,Z -51.065,A -90.000,B 90.000,C 0.000} C_DIS
LIN {X 63.430,Y -25.345,Z -52.210,A -90.000,B 90.000,C 0.000} C_DIS
LIN {X 64.546,Y -25.350,Z -53.168,A -90.000,B 90.000,C 0.000} C_DIS
LIN {X 65.143,Y -25.352,Z -53.696,A -90.000,B 90.000,C 0.000} C_DIS
LIN {X 65.281,Y -25.355,Z -53.797,A -90.000,B 90.000,C 0.000} C_DIS
LIN {X 65.888,Y -25.358,Z -54.242,A -90.000,B 90.000,C 0.000} C_DIS
LIN {X 66.397,Y -25.363,Z -54.599,A -90.000,B 90.000,C 0.000} C_DIS
LIN {X 67.106,Y -25.368,Z -55.095,A -90.000,B 90.000,C 0.000} C_DIS
LIN {X 67.414,Y -25.371,Z -55.299,A -90.000,B 90.000,C 0.000} C_DIS
LIN {X 68.034,Y -25.378,Z -55.694,A -90.000,B 90.000,C 0.000} C_DIS
LIN {X 68.809,Y -25.383,Z -56.188,A -90.000,B 90.000,C 0.000} C_DIS
LIN {X 69.269,Y -25.385,Z -56.487,A -90.000,B 90.000,C 0.000} C_DIS
LIN {X 70.843,Y -25.406,Z -57.499,A -90.000,B 90.000,C 0.000} C_DIS
LIN {X 71.243,Y -25.409,Z -57.758,A -90.000,B 90.000,C 0.000} C_DIS
LIN {X 71.440,Y -25.406,Z -57.903,A -90.000,B 90.000,C 0.000} C_DIS
LIN {X 71.833,Y -25.411,Z -58.194,A -90.000,B 90.000,C 0.000} C_DIS
LIN {X 73.108,Y -25.432,Z -59.117,A -90.000,B 90.000,C 0.000} C_DIS
LIN {X 73.479,Y -25.429,Z -59.415,A -90.000,B 90.000,C 0.000} C_DIS
LIN {X 73.640,Y -25.426,Z -59.560,A -90.000,B 90.000,C 0.000} C_DIS
LIN {X 74.219,Y -25.434,Z -60.092,A -90.000,B 90.000,C 0.000} C_DIS
LIN {X 74.389,Y -25.435,Z -60.255,A -90.000,B 90.000,C 0.000} C_DIS
LIN {X 75.003,Y -25.443,Z -60.849,A -90.000,B 90.000,C 0.000} C_DIS
LIN {X 75.340,Y -25.445,Z -61.186,A -90.000,B 90.000,C 0.000} C_DIS
LIN {X 75.477,Y -25.442,Z -61.339,A -90.000,B 90.000,C 0.000} C_DIS
LIN {X 75.641,Y -25.444,Z -61.526,A -90.000,B 90.000,C 0.000} C_DIS
LIN {X 75.828,Y -25.445,Z -61.749,A -90.000,B 90.000,C 0.000} C_DIS
LIN {X 76.797,Y -25.464,Z -62.921,A -90.000,B 90.000,C 0.000} C_DIS
LIN {X 77.048,Y -25.462,Z -63.259,A -90.000,B 90.000,C 0.000} C_DIS
LIN {X 77.113,Y -25.464,Z -63.349,A -90.000,B 90.000,C 0.000} C_DIS
LIN {X 77.827,Y -25.475,Z -64.382,A -90.000,B 90.000,C 0.000} C_DIS
LIN {X 78.100,Y -25.474,Z -64.792,A -90.000,B 90.000,C 0.000} C_DIS
LIN {X 78.318,Y -25.377,Z -65.060,A -90.000,B 90.000,C 0.000} C_DIS
LIN {X 78.477,Y -25.332,Z -65.279,A -90.000,B 90.000,C 0.000} C_DIS
LIN {X 78.538,Y -25.321,Z -65.365,A -90.000,B 90.000,C 0.000} C_DIS
LIN {X 79.023,Y -25.318,Z -63.714,A -90.000,B 90.000,C 0.000} C_DIS
LIN {X 79.744,Y -25.318,Z -61.550,A -90.000,B 90.000,C 0.000} C_DIS
LIN {X 79.787,Y -25.318,Z -61.437,A -90.000,B 90.000,C 0.000} C_DIS
LIN {X 80.297,Y -25.329,Z -59.799,A -90.000,B 90.000,C 0.000} C_DIS
LIN {X 80.458,Y -25.332,Z -59.321,A -90.000,B 90.000,C 0.000} C_DIS
LIN {X 80.594,Y -25.335,Z -58.952,A -90.000,B 90.000,C 0.000} C_DIS
LIN {X 81.205,Y -25.331,Z -57.294,A -90.000,B 90.000,C 0.000} C_DIS
LIN {X 81.757,Y -25.327,Z -56.054,A -90.000,B 90.000,C 0.000} C_DIS
LIN {X 82.142,Y -25.329,Z -55.094,A -90.000,B 90.000,C 0.000} C_DIS
LIN {X 82.335,Y -25.332,Z -54.668,A -90.000,B 90.000,C 0.000} C_DIS
LIN {X 83.333,Y -25.328,Z -52.807,A -90.000,B 90.000,C 0.000} C_DIS
LIN {X 83.588,Y -25.329,Z -52.374,A -90.000,B 90.000,C 0.000} C_DIS
LIN {X 84.750,Y -25.320,Z -50.668,A -90.000,B 90.000,C 0.000} C_DIS
LIN {X 85.030,Y -25.320,Z -50.285,A -90.000,B 90.000,C 0.000} C_DIS
LIN {X 86.348,Y -25.311,Z -48.702,A -90.000,B 90.000,C 0.000} C_DIS
LIN {X 86.674,Y -25.311,Z -48.342,A -90.000,B 90.000,C 0.000} C_DIS
LIN {X 88.117,Y -25.309,Z -46.880,A -90.000,B 90.000,C 0.000} C_DIS
LIN {X 88.495,Y -25.309,Z -46.539,A -90.000,B 90.000,C 0.000} C_DIS
LIN {X 89.960,Y -25.320,Z -45.253,A -90.000,B 90.000,C 0.000} C_DIS
LIN {X 90.061,Y -25.308,Z -45.164,A -90.000,B 90.000,C 0.000} C_DIS
LIN {X 90.061,Y -60.000,Z -45.164,A -90.000,B 90.000,C 0.000} C_DIS
LIN {X 116.506,Y -60.000,Z -47.954,A -90.000,B 90.000,C 0.000} C_DIS
LIN {X 116.506,Y -25.308,Z -47.954,A -90.000,B 90.000,C 0.000} C_DIS
LIN {X 116.372,Y -25.308,Z -48.278,A -90.000,B 90.000,C 0.000} C_DIS
LIN {X 116.294,Y -25.308,Z -48.466,A -90.000,B 90.000,C 0.000} C_DIS
LIN {X 116.211,Y -25.308,Z -48.654,A -90.000,B 90.000,C 0.000} C_DIS
LIN {X 116.177,Y -25.308,Z -48.721,A -90.000,B 90.000,C 0.000} C_DIS
LIN {X 116.166,Y -25.308,Z -48.738,A -90.000,B 90.000,C 0.000} C_DIS
LIN {X 116.156,Y -25.308,Z -48.745,A -90.000,B 90.000,C 0.000} C_DIS
LIN {X 116.162,Y -25.308,Z -48.741,A -90.000,B 90.000,C 0.000} C_DIS
LIN {X 116.162,Y -25.307,Z -48.731,A -90.000,B 90.000,C 0.000} C_DIS
LIN {X 116.173,Y -25.308,Z -48.707,A -90.000,B 90.000,C 0.000} C_DIS
LIN {X 116.173,Y -35.308,Z -48.706,A -90.000,B 90.000,C 0.000} C_DIS
LIN {X 116.175,Y -35.622,Z -48.699,A -90.000,B 90.000,C 0.000} C_DIS
LIN {X 116.178,Y -35.718,Z -48.683,A -90.000,B 90.000,C 0.000} C_DIS
LIN {X 116.188,Y -35.846,Z -48.646,A -90.000,B 90.000,C 0.000} C_DIS
LIN {X 116.216,Y -36.039,Z -48.549,A -90.000,B 90.000,C 0.000} C_DIS
LIN {X 116.254,Y -36.204,Z -48.425,A -90.000,B 90.000,C 0.000} C_DIS
LIN {X 116.301,Y -36.351,Z -48.277,A -90.000,B 90.000,C 0.000} C_DIS
LIN {X 116.356,Y -36.460,Z -48.108,A -90.000,B 90.000,C 0.000} C_DIS
LIN {X 116.418,Y -36.546,Z -47.923,A -90.000,B 90.000,C 0.000} C_DIS
LIN {X 116.558,Y -36.717,Z -47.516,A -90.000,B 90.000,C 0.000} C_DIS
LIN {X 116.710,Y -36.871,Z -47.082,A -90.000,B 90.000,C 0.000} C_DIS
LIN {X 116.787,Y -36.886,Z -46.863,A -90.000,B 90.000,C 0.000} C_DIS
LIN {X 116.864,Y -36.874,Z -46.649,A -90.000,B 90.000,C 0.000} C_DIS
LIN {X 117.012,Y -36.837,Z -46.244,A -90.000,B 90.000,C 0.000} C_DIS
LIN {X 117.080,Y -36.806,Z -46.061,A -90.000,B 90.000,C 0.000} C_DIS
LIN {X 117.143,Y -36.735,Z -45.896,A -90.000,B 90.000,C 0.000} C_DIS
LIN {X 117.200,Y -36.633,Z -45.751,A -90.000,B 90.000,C 0.000} C_DIS
LIN {X 117.248,Y -36.508,Z -45.630,A -90.000,B 90.000,C 0.000} C_DIS
LIN {X 117.288,Y -36.352,Z -45.537,A -90.000,B 90.000,C 0.000} C_DIS
LIN {X 117.304,Y -36.250,Z -45.503,A -90.000,B 90.000,C 0.000} C_DIS
LIN {X 117.317,Y -36.098,Z -45.476,A -90.000,B 90.000,C 0.000} C_DIS
LIN {X 117.320,Y -36.031,Z -45.471,A -90.000,B 90.000,C 0.000} C_DIS
LIN {X 117.321,Y -25.306,Z -45.468,A -90.000,B 90.000,C 0.000} C_DIS
LIN {X 117.327,Y -25.308,Z -45.447,A -90.000,B 90.000,C 0.000} C_DIS
LIN {X 117.325,Y -25.307,Z -45.451,A -90.000,B 90.000,C 0.000} C_DIS
LIN {X 117.328,Y -25.308,Z -45.442,A -90.000,B 90.000,C 0.000} C_DIS
LIN {X 117.326,Y -25.308,Z -45.472,A -90.000,B 90.000,C 0.000} C_DIS
LIN {X 117.320,Y -25.308,Z -45.504,A -90.000,B 90.000,C 0.000} C_DIS
LIN {X 117.264,Y -25.306,Z -45.746,A -90.000,B 90.000,C 0.000} C_DIS
LIN {X 117.200,Y -25.308,Z -45.940,A -90.000,B 90.000,C 0.000} C_DIS
LIN {X 117.121,Y -25.308,Z -46.207,A -90.000,B 90.000,C 0.000} C_DIS
LIN {X 117.121,Y -60.000,Z -46.207,A -90.000,B 90.000,C 0.000} C_DIS
LIN {X 101.846,Y -60.000,Z -82.605,A -90.000,B 90.000,C 0.000} C_DIS
LIN {X 101.846,Y -25.308,Z -82.605,A -90.000,B 90.000,C 0.000} C_DIS
LIN {X 101.717,Y -25.322,Z -82.799,A -90.000,B 90.000,C 0.000} C_DIS
LIN {X 101.429,Y -25.308,Z -83.230,A -90.000,B 90.000,C 0.000} C_DIS
LIN {X 101.429,Y -60.000,Z -83.230,A -90.000,B 90.000,C 0.000} C_DIS
LIN {X 16.086,Y -60.000,Z -52.149,A -90.000,B 90.000,C 0.000} C_DIS
LIN {X 16.086,Y -25.308,Z -52.149,A -90.000,B 90.000,C 0.000} C_DIS
LIN {X 16.213,Y -25.363,Z -52.142,A -90.000,B 90.000,C 0.000} C_DIS
LIN {X 16.390,Y -25.443,Z -52.140,A -90.000,B 90.000,C 0.000} C_DIS
LIN {X 16.520,Y -25.490,Z -52.103,A -90.000,B 90.000,C 0.000} C_DIS
LIN {X 16.722,Y -25.566,Z -52.058,A -90.000,B 90.000,C 0.000} C_DIS
LIN {X 16.952,Y -25.656,Z -52.016,A -90.000,B 90.000,C 0.000} C_DIS
LIN {X 17.252,Y -25.773,Z -51.970,A -90.000,B 90.000,C 0.000} C_DIS
LIN {X 17.406,Y -25.835,Z -51.951,A -90.000,B 90.000,C 0.000} C_DIS
LIN {X 17.445,Y -25.823,Z -51.866,A -90.000,B 90.000,C 0.000} C_DIS
LIN {X 17.549,Y -25.787,Z -51.645,A -90.000,B 90.000,C 0.000} C_DIS
LIN {X 17.636,Y -25.754,Z -51.461,A -90.000,B 90.000,C 0.000} C_DIS
LIN {X 17.804,Y -25.691,Z -51.126,A -90.000,B 90.000,C 0.000} C_DIS
LIN {X 17.860,Y -25.671,Z -51.024,A -90.000,B 90.000,C 0.000} C_DIS
LIN {X 17.926,Y -25.651,Z -50.912,A -90.000,B 90.000,C 0.000} C_DIS
LIN {X 17.989,Y -25.633,Z -50.809,A -90.000,B 90.000,C 0.000} C_DIS
LIN {X 18.097,Y -25.610,Z -50.649,A -90.000,B 90.000,C 0.000} C_DIS
LIN {X 18.237,Y -25.584,Z -50.452,A -90.000,B 90.000,C 0.000} C_DIS
LIN {X 18.309,Y -25.570,Z -50.355,A -90.000,B 90.000,C 0.000} C_DIS
LIN {X 18.578,Y -25.505,Z -50.002,A -90.000,B 90.000,C 0.000} C_DIS
LIN {X 18.760,Y -25.452,Z -49.771,A -90.000,B 90.000,C 0.000} C_DIS
LIN {X 18.887,Y -25.420,Z -49.621,A -90.000,B 90.000,C 0.000} C_DIS
LIN {X 18.977,Y -25.403,Z -49.516,A -90.000,B 90.000,C 0.000} C_DIS
LIN {X 19.136,Y -25.364,Z -49.321,A -90.000,B 90.000,C 0.000} C_DIS
LIN {X 19.242,Y -25.339,Z -49.201,A -90.000,B 90.000,C 0.000} C_DIS
LIN {X 19.394,Y -25.308,Z -49.037,A -90.000,B 90.000,C 0.000} C_DIS
LIN {X 19.394,Y -60.000,Z -49.037,A -90.000,B 90.000,C 0.000} C_DIS
LIN {X -88.319,Y -60.000,Z -44.460,A -90.000,B 90.000,C 0.000} C_DIS
LIN {X -88.319,Y -25.308,Z -44.460,A -90.000,B 90.000,C 0.000} C_DIS
LIN {X -88.092,Y -25.358,Z -44.495,A -90.000,B 90.000,C 0.000} C_DIS
LIN {X -87.820,Y -25.417,Z -44.541,A -90.000,B 90.000,C 0.000} C_DIS
LIN {X -87.508,Y -25.486,Z -44.598,A -90.000,B 90.000,C 0.000} C_DIS
LIN {X -87.286,Y -25.534,Z -44.648,A -90.000,B 90.000,C 0.000} C_DIS
LIN {X -86.917,Y -25.610,Z -44.752,A -90.000,B 90.000,C 0.000} C_DIS
LIN {X -86.738,Y -25.647,Z -44.809,A -90.000,B 90.000,C 0.000} C_DIS
LIN {X -86.219,Y -25.753,Z -44.985,A -90.000,B 90.000,C 0.000} C_DIS
LIN {X -85.906,Y -25.817,Z -45.101,A -90.000,B 90.000,C 0.000} C_DIS
LIN {X -85.568,Y -25.885,Z -45.232,A -90.000,B 90.000,C 0.000} C_DIS
LIN {X -85.146,Y -25.969,Z -45.407,A -90.000,B 90.000,C 0.000} C_DIS
LIN {X -84.809,Y -26.033,Z -45.556,A -90.000,B 90.000,C 0.000} C_DIS
LIN {X -84.397,Y -26.106,Z -45.743,A -90.000,B 90.000,C 0.000} C_DIS
LIN {X -84.316,Y -26.120,Z -45.781,A -90.000,B 90.000,C 0.000} C_DIS
LIN {X -84.120,Y -26.158,Z -45.829,A -90.000,B 90.000,C 0.000} C_DIS
LIN {X -83.827,Y -26.214,Z -45.904,A -90.000,B 90.000,C 0.000} C_DIS
LIN {X -83.684,Y -26.240,Z -45.946,A -90.000,B 90.000,C 0.000} C_DIS
LIN {X -83.538,Y -26.267,Z -45.993,A -90.000,B 90.000,C 0.000} C_DIS
LIN {X -83.010,Y -26.364,Z -46.171,A -90.000,B 90.000,C 0.000} C_DIS
LIN {X -82.652,Y -26.418,Z -46.290,A -90.000,B 90.000,C 0.000} C_DIS
LIN {X -82.393,Y -26.457,Z -46.383,A -90.000,B 90.000,C 0.000} C_DIS
LIN {X -81.680,Y -26.573,Z -46.648,A -90.000,B 90.000,C 0.000} C_DIS
LIN {X -81.388,Y -26.620,Z -46.762,A -90.000,B 90.000,C 0.000} C_DIS
LIN {X -81.205,Y -26.649,Z -46.840,A -90.000,B 90.000,C 0.000} C_DIS
LIN {X -80.886,Y -26.694,Z -46.994,A -90.000,B 90.000,C 0.000} C_DIS
LIN {X -80.329,Y -26.763,Z -47.264,A -90.000,B 90.000,C 0.000} C_DIS
LIN {X -80.024,Y -26.800,Z -47.418,A -90.000,B 90.000,C 0.000} C_DIS
LIN {X -79.687,Y -26.842,Z -47.584,A -90.000,B 90.000,C 0.000} C_DIS
LIN {X -79.656,Y -26.865,Z -47.387,A -90.000,B 90.000,C 0.000} C_DIS
LIN {X -79.647,Y -26.870,Z -47.343,A -90.000,B 90.000,C 0.000} C_DIS
LIN {X -79.640,Y -26.891,Z -47.123,A -90.000,B 90.000,C 0.000} C_DIS
LIN {X -79.628,Y -26.903,Z -46.942,A -90.000,B 90.000,C 0.000} C_DIS
LIN {X -79.615,Y -26.910,Z -46.797,A -90.000,B 90.000,C 0.000} C_DIS
LIN {X -79.603,Y -26.914,Z -46.706,A -90.000,B 90.000,C 0.000} C_DIS
LIN {X -79.583,Y -26.921,Z -46.579,A -90.000,B 90.000,C 0.000} C_DIS
LIN {X -79.565,Y -26.927,Z -46.486,A -90.000,B 90.000,C 0.000} C_DIS
LIN {X -79.517,Y -26.941,Z -46.269,A -90.000,B 90.000,C 0.000} C_DIS
LIN {X -79.462,Y -26.956,Z -46.076,A -90.000,B 90.000,C 0.000} C_DIS
LIN {X -79.411,Y -26.969,Z -45.923,A -90.000,B 90.000,C 0.000} C_DIS
LIN {X -79.339,Y -26.985,Z -45.741,A -90.000,B 90.000,C 0.000} C_DIS
LIN {X -79.298,Y -26.989,Z -45.640,A -90.000,B 90.000,C 0.000} C_DIS
LIN {X -79.263,Y -26.992,Z -45.564,A -90.000,B 90.000,C 0.000} C_DIS
LIN {X -79.196,Y -26.995,Z -45.438,A -90.000,B 90.000,C 0.000} C_DIS
LIN {X -79.079,Y -26.995,Z -45.225,A -90.000,B 90.000,C 0.000} C_DIS
LIN {X -79.036,Y -26.995,Z -45.154,A -90.000,B 90.000,C 0.000} C_DIS
LIN {X -78.886,Y -26.996,Z -44.932,A -90.000,B 90.000,C 0.000} C_DIS
LIN {X -78.815,Y -26.995,Z -44.835,A -90.000,B 90.000,C 0.000} C_DIS
LIN {X -78.741,Y -26.993,Z -44.740,A -90.000,B 90.000,C 0.000} C_DIS
LIN {X -78.627,Y -26.990,Z -44.601,A -90.000,B 90.000,C 0.000} C_DIS
LIN {X -78.516,Y -26.988,Z -44.479,A -90.000,B 90.000,C 0.000} C_DIS
LIN {X -78.386,Y -26.986,Z -44.349,A -90.000,B 90.000,C 0.000} C_DIS
LIN {X -78.305,Y -26.983,Z -44.271,A -90.000,B 90.000,C 0.000} C_DIS
LIN {X -78.165,Y -26.976,Z -44.150,A -90.000,B 90.000,C 0.000} C_DIS
LIN {X -78.073,Y -26.972,Z -44.077,A -90.000,B 90.000,C 0.000} C_DIS
LIN {X -77.910,Y -26.966,Z -43.955,A -90.000,B 90.000,C 0.000} C_DIS
LIN {X -77.858,Y -26.962,Z -43.920,A -90.000,B 90.000,C 0.000} C_DIS
LIN {X -77.729,Y -26.949,Z -43.837,A -90.000,B 90.000,C 0.000} C_DIS
LIN {X -77.552,Y -26.932,Z -43.734,A -90.000,B 90.000,C 0.000} C_DIS
LIN {X -77.376,Y -26.913,Z -43.644,A -90.000,B 90.000,C 0.000} C_DIS
LIN {X -77.265,Y -26.901,Z -43.593,A -90.000,B 90.000,C 0.000} C_DIS
LIN {X -77.146,Y -26.889,Z -43.544,A -90.000,B 90.000,C 0.000} C_DIS
LIN {X -76.954,Y -26.867,Z -43.468,A -90.000,B 90.000,C 0.000} C_DIS
LIN {X -76.777,Y -26.848,Z -43.407,A -90.000,B 90.000,C 0.000} C_DIS
LIN {X -76.286,Y -26.797,Z -43.244,A -90.000,B 90.000,C 0.000} C_DIS
LIN {X -76.130,Y -26.775,Z -43.193,A -90.000,B 90.000,C 0.000} C_DIS
LIN {X -75.915,Y -26.744,Z -43.128,A -90.000,B 90.000,C 0.000} C_DIS
LIN {X -75.791,Y -26.727,Z -43.096,A -90.000,B 90.000,C 0.000} C_DIS
LIN {X -75.415,Y -26.681,Z -43.013,A -90.000,B 90.000,C 0.000} C_DIS
LIN {X -75.336,Y -26.673,Z -42.997,A -90.000,B 90.000,C 0.000} C_DIS
LIN {X -75.018,Y -26.636,Z -42.948,A -90.000,B 90.000,C 0.000} C_DIS
LIN {X -74.801,Y -26.613,Z -42.929,A -90.000,B 90.000,C 0.000} C_DIS
LIN {X -74.617,Y -26.597,Z -42.923,A -90.000,B 90.000,C 0.000} C_DIS
LIN {X -74.389,Y -26.580,Z -42.927,A -90.000,B 90.000,C 0.000} C_DIS
LIN {X -74.107,Y -26.562,Z -42.942,A -90.000,B 90.000,C 0.000} C_DIS
LIN {X -73.985,Y -26.555,Z -42.952,A -90.000,B 90.000,C 0.000} C_DIS
LIN {X -73.803,Y -26.545,Z -42.973,A -90.000,B 90.000,C 0.000} C_DIS
LIN {X -73.630,Y -26.538,Z -43.003,A -90.000,B 90.000,C 0.000} C_DIS
LIN {X -72.405,Y -26.473,Z -43.156,A -90.000,B 90.000,C 0.000} C_DIS
LIN {X -72.330,Y -26.468,Z -43.168,A -90.000,B 90.000,C 0.000} C_DIS
LIN {X -72.150,Y -26.460,Z -43.205,A -90.000,B 90.000,C 0.000} C_DIS
LIN {X -71.856,Y -26.451,Z -43.279,A -90.000,B 90.000,C 0.000} C_DIS
LIN {X -71.768,Y -26.449,Z -43.303,A -90.000,B 90.000,C 0.000} C_DIS
LIN {X -71.516,Y -26.447,Z -43.387,A -90.000,B 90.000,C 0.000} C_DIS
LIN {X -70.850,Y -26.422,Z -43.545,A -90.000,B 90.000,C 0.000} C_DIS
LIN {X -70.457,Y -26.401,Z -43.641,A -90.000,B 90.000,C 0.000} C_DIS
LIN {X -70.283,Y -26.394,Z -43.689,A -90.000,B 90.000,C 0.000} C_DIS
LIN {X -69.939,Y -26.385,Z -43.803,A -90.000,B 90.000,C 0.000} C_DIS
LIN {X -69.124,Y -26.339,Z -44.000,A -90.000,B 90.000,C 0.000} C_DIS
LIN {X -69.025,Y -26.329,Z -44.011,A -90.000,B 90.000,C 0.000} C_DIS
LIN {X -68.779,Y -26.303,Z -44.046,A -90.000,B 90.000,C 0.000} C_DIS
LIN {X -68.679,Y -26.294,Z -44.065,A -90.000,B 90.000,C 0.000} C_DIS
LIN {X -67.394,Y -26.190,Z -44.350,A -90.000,B 90.000,C 0.000} C_DIS
LIN {X -67.228,Y -26.176,Z -44.387,A -90.000,B 90.000,C 0.000} C_DIS
LIN {X -66.751,Y -26.134,Z -44.487,A -90.000,B 90.000,C 0.000} C_DIS
LIN {X -66.672,Y -26.128,Z -44.504,A -90.000,B 90.000,C 0.000} C_DIS
LIN {X -66.158,Y -26.073,Z -44.580,A -90.000,B 90.000,C 0.000} C_DIS
LIN {X -65.940,Y -26.053,Z -44.622,A -90.000,B 90.000,C 0.000} C_DIS
LIN {X -65.674,Y -26.031,Z -44.684,A -90.000,B 90.000,C 0.000} C_DIS
LIN {X -64.539,Y -25.937,Z -44.955,A -90.000,B 90.000,C 0.000} C_DIS
LIN {X -64.353,Y -25.925,Z -44.998,A -90.000,B 90.000,C 0.000} C_DIS
LIN {X -64.167,Y -25.907,Z -45.027,A -90.000,B 90.000,C 0.000} C_DIS
LIN {X -63.861,Y -25.879,Z -45.084,A -90.000,B 90.000,C 0.000} C_DIS
LIN {X -63.183,Y -25.819,Z -45.216,A -90.000,B 90.000,C 0.000} C_DIS
LIN {X -62.907,Y -25.797,Z -45.279,A -90.000,B 90.000,C 0.000} C_DIS
LIN {X -62.216,Y -25.749,Z -45.453,A -90.000,B 90.000,C 0.000} C_DIS
LIN {X -61.529,Y -25.716,Z -45.620,A -90.000,B 90.000,C 0.000} C_DIS
LIN {X -61.180,Y -25.689,Z -45.679,A -90.000,B 90.000,C 0.000} C_DIS
LIN {X -61.005,Y -25.677,Z -45.714,A -90.000,B 90.000,C 0.000} C_DIS
LIN {X -59.955,Y -25.619,Z -45.953,A -90.000,B 90.000,C 0.000} C_DIS
LIN {X -59.620,Y -25.603,Z -46.038,A -90.000,B 90.000,C 0.000} C_DIS
LIN {X -58.634,Y -25.588,Z -46.276,A -90.000,B 90.000,C 0.000} C_DIS
LIN {X -58.004,Y -25.566,Z -46.397,A -90.000,B 90.000,C 0.000} C_DIS
LIN {X -57.625,Y -25.559,Z -46.484,A -90.000,B 90.000,C 0.000} C_DIS
LIN {X -56.960,Y -25.544,Z -46.644,A -90.000,B 90.000,C 0.000} C_DIS
LIN {X -55.811,Y -25.548,Z -46.915,A -90.000,B 90.000,C 0.000} C_DIS
LIN {X -55.585,Y -25.549,Z -46.967,A -90.000,B 90.000,C 0.000} C_DIS
LIN {X -54.537,Y -25.538,Z -47.180,A -90.000,B 90.000,C 0.000} C_DIS
LIN {X -54.259,Y -25.536,Z -47.245,A -90.000,B 90.000,C 0.000} C_DIS
LIN {X -53.648,Y -25.550,Z -47.383,A -90.000,B 90.000,C 0.000} C_DIS
LIN {X -53.138,Y -25.561,Z -47.496,A -90.000,B 90.000,C 0.000} C_DIS
LIN {X -52.543,Y -25.572,Z -47.629,A -90.000,B 90.000,C 0.000} C_DIS
LIN {X -51.369,Y -25.585,Z -47.885,A -90.000,B 90.000,C 0.000} C_DIS
LIN {X -50.817,Y -25.603,Z -48.001,A -90.000,B 90.000,C 0.000} C_DIS
LIN {X -50.513,Y -25.611,Z -48.066,A -90.000,B 90.000,C 0.000} C_DIS
LIN {X -50.216,Y -25.622,Z -48.135,A -90.000,B 90.000,C 0.000} C_DIS
LIN {X -49.571,Y -25.635,Z -48.291,A -90.000,B 90.000,C 0.000} C_DIS
LIN {X -48.679,Y -25.646,Z -48.492,A -90.000,B 90.000,C 0.000} C_DIS
LIN {X -48.341,Y -25.653,Z -48.574,A -90.000,B 90.000,C 0.000} C_DIS
LIN {X -47.453,Y -25.682,Z -48.784,A -90.000,B 90.000,C 0.000} C_DIS
LIN {X -46.919,Y -25.692,Z -48.897,A -90.000,B 90.000,C 0.000} C_DIS
LIN {X -46.657,Y -25.699,Z -48.956,A -90.000,B 90.000,C 0.000} C_DIS
LIN {X -46.557,Y -25.697,Z -48.969,A -90.000,B 90.000,C 0.000} C_DIS
LIN {X -45.907,Y -25.653,Z -49.010,A -90.000,B 90.000,C 0.000} C_DIS
LIN {X -45.347,Y -25.617,Z -49.050,A -90.000,B 90.000,C 0.000} C_DIS
LIN {X -44.879,Y -25.591,Z -49.080,A -90.000,B 90.000,C 0.000} C_DIS
LIN {X -44.277,Y -25.552,Z -49.116,A -90.000,B 90.000,C 0.000} C_DIS
LIN {X -43.784,Y -25.516,Z -49.148,A -90.000,B 90.000,C 0.000} C_DIS
LIN {X -43.244,Y -25.483,Z -49.194,A -90.000,B 90.000,C 0.000} C_DIS
LIN {X -42.567,Y -25.437,Z -49.254,A -90.000,B 90.000,C 0.000} C_DIS
LIN {X -42.116,Y -25.416,Z -49.306,A -90.000,B 90.000,C 0.000} C_DIS
LIN {X -41.457,Y -25.389,Z -49.385,A -90.000,B 90.000,C 0.000} C_DIS
LIN {X -39.703,Y -25.314,Z -49.610,A -90.000,B 90.000,C 0.000} C_DIS
LIN {X -39.593,Y -25.308,Z -49.625,A -90.000,B 90.000,C 0.000} C_DIS
LIN {X -39.593,Y -60.000,Z -49.625,A -90.000,B 90.000,C 0.000} C_DIS
LIN {X -88.340,Y -60.000,Z -42.460,A -90.000,B 90.000,C 0.000} C_DIS
LIN {X -88.340,Y -25.308,Z -42.460,A -90.000,B 90.000,C 0.000} C_DIS
LIN {X -88.031,Y -25.386,Z -42.482,A -90.000,B 90.000,C 0.000} C_DIS
LIN {X -87.647,Y -25.484,Z -42.544,A -90.000,B 90.000,C 0.000} C_DIS
LIN {X -87.366,Y -25.556,Z -42.594,A -90.000,B 90.000,C 0.000} C_DIS
LIN {X -87.173,Y -25.604,Z -42.629,A -90.000,B 90.000,C 0.000} C_DIS
LIN {X -86.915,Y -25.667,Z -42.687,A -90.000,B 90.000,C 0.000} C_DIS
LIN {X -86.779,Y -25.700,Z -42.720,A -90.000,B 90.000,C 0.000} C_DIS
LIN {X -86.353,Y -25.805,Z -42.843,A -90.000,B 90.000,C 0.000} C_DIS
LIN {X -86.197,Y -25.844,Z -42.894,A -90.000,B 90.000,C 0.000} C_DIS
LIN {X -85.898,Y -25.918,Z -42.996,A -90.000,B 90.000,C 0.000} C_DIS
LIN {X -85.570,Y -25.992,Z -43.109,A -90.000,B 90.000,C 0.000} C_DIS
LIN {X -85.237,Y -26.066,Z -43.233,A -90.000,B 90.000,C 0.000} C_DIS
LIN {X -84.852,Y -26.142,Z -43.382,A -90.000,B 90.000,C 0.000} C_DIS
LIN {X -84.378,Y -26.235,Z -43.579,A -90.000,B 90.000,C 0.000} C_DIS
LIN {X -83.966,Y -26.315,Z -43.763,A -90.000,B 90.000,C 0.000} C_DIS
LIN {X -83.700,Y -26.366,Z -43.885,A -90.000,B 90.000,C 0.000} C_DIS
LIN {X -83.315,Y -26.441,Z -43.984,A -90.000,B 90.000,C 0.000} C_DIS
LIN {X -83.076,Y -26.483,Z -44.055,A -90.000,B 90.000,C 0.000} C_DIS
LIN {X -82.826,Y -26.528,Z -44.138,A -90.000,B 90.000,C 0.000} C_DIS
LIN {X -82.013,Y -26.639,Z -44.408,A -90.000,B 90.000,C 0.000} C_DIS
LIN {X -81.732,Y -26.681,Z -44.509,A -90.000,B 90.000,C 0.000} C_DIS
LIN {X -81.078,Y -26.781,Z -44.751,A -90.000,B 90.000,C 0.000} C_DIS
LIN {X -81.042,Y -26.788,Z -44.674,A -90.000,B 90.000,C 0.000} C_DIS
LIN {X -80.889,Y -26.801,Z -44.386,A -90.000,B 90.000,C 0.000} C_DIS
LIN {X -80.783,Y -26.810,Z -44.195,A -90.000,B 90.000,C 0.000} C_DIS
LIN {X -80.671,Y -26.819,Z -44.015,A -90.000,B 90.000,C 0.000} C_DIS
LIN {X -80.599,Y -26.825,Z -43.908,A -90.000,B 90.000,C 0.000} C_DIS
LIN {X -80.505,Y -26.826,Z -43.771,A -90.000,B 90.000,C 0.000} C_DIS
LIN {X -80.426,Y -26.826,Z -43.662,A -90.000,B 90.000,C 0.000} C_DIS
LIN {X -80.329,Y -26.823,Z -43.535,A -90.000,B 90.000,C 0.000} C_DIS
LIN {X -80.176,Y -26.811,Z -43.348,A -90.000,B 90.000,C 0.000} C_DIS
LIN {X -80.105,Y -26.805,Z -43.267,A -90.000,B 90.000,C 0.000} C_DIS
LIN {X -79.980,Y -26.796,Z -43.130,A -90.000,B 90.000,C 0.000} C_DIS
LIN {X -79.888,Y -26.790,Z -43.036,A -90.000,B 90.000,C 0.000} C_DIS
LIN {X -79.766,Y -26.776,Z -42.916,A -90.000,B 90.000,C 0.000} C_DIS
LIN {X -79.684,Y -26.765,Z -42.839,A -90.000,B 90.000,C 0.000} C_DIS
LIN {X -79.613,Y -26.756,Z -42.775,A -90.000,B 90.000,C 0.000} C_DIS
LIN {X -79.410,Y -26.733,Z -42.604,A -90.000,B 90.000,C 0.000} C_DIS
LIN {X -79.264,Y -26.717,Z -42.490,A -90.000,B 90.000,C 0.000} C_DIS
LIN {X -79.033,Y -26.688,Z -42.324,A -90.000,B 90.000,C 0.000} C_DIS
LIN {X -78.807,Y -26.661,Z -42.177,A -90.000,B 90.000,C 0.000} C_DIS
LIN {X -78.721,Y -26.648,Z -42.126,A -90.000,B 90.000,C 0.000} C_DIS
LIN {X -78.566,Y -26.617,Z -42.039,A -90.000,B 90.000,C 0.000} C_DIS
LIN {X -78.446,Y -26.594,Z -41.977,A -90.000,B 90.000,C 0.000} C_DIS
LIN {X -78.287,Y -26.564,Z -41.898,A -90.000,B 90.000,C 0.000} C_DIS
LIN {X -78.047,Y -26.523,Z -41.792,A -90.000,B 90.000,C 0.000} C_DIS
LIN {X -77.904,Y -26.498,Z -41.734,A -90.000,B 90.000,C 0.000} C_DIS
LIN {X -77.714,Y -26.465,Z -41.662,A -90.000,B 90.000,C 0.000} C_DIS
LIN {X -77.574,Y -26.442,Z -41.613,A -90.000,B 90.000,C 0.000} C_DIS
LIN {X -77.076,Y -26.355,Z -41.455,A -90.000,B 90.000,C 0.000} C_DIS
LIN {X -76.760,Y -26.299,Z -41.355,A -90.000,B 90.000,C 0.000} C_DIS
LIN {X -76.574,Y -26.266,Z -41.301,A -90.000,B 90.000,C 0.000} C_DIS
LIN {X -76.442,Y -26.240,Z -41.265,A -90.000,B 90.000,C 0.000} C_DIS
LIN {X -76.266,Y -26.208,Z -41.224,A -90.000,B 90.000,C 0.000} C_DIS
LIN {X -75.994,Y -26.159,Z -41.169,A -90.000,B 90.000,C 0.000} C_DIS
LIN {X -75.830,Y -26.128,Z -41.137,A -90.000,B 90.000,C 0.000} C_DIS
LIN {X -75.697,Y -26.104,Z -41.114,A -90.000,B 90.000,C 0.000} C_DIS
LIN {X -75.412,Y -26.054,Z -41.075,A -90.000,B 90.000,C 0.000} C_DIS
LIN {X -75.290,Y -26.035,Z -41.060,A -90.000,B 90.000,C 0.000} C_DIS
LIN {X -75.025,Y -25.998,Z -41.040,A -90.000,B 90.000,C 0.000} C_DIS
LIN {X -74.878,Y -25.980,Z -41.033,A -90.000,B 90.000,C 0.000} C_DIS
LIN {X -74.694,Y -25.959,Z -41.029,A -90.000,B 90.000,C 0.000} C_DIS
LIN {X -74.631,Y -25.952,Z -41.030,A -90.000,B 90.000,C 0.000} C_DIS
LIN {X -74.329,Y -25.923,Z -41.039,A -90.000,B 90.000,C 0.000} C_DIS
LIN {X -73.998,Y -25.895,Z -41.060,A -90.000,B 90.000,C 0.000} C_DIS
LIN {X -73.799,Y -25.880,Z -41.078,A -90.000,B 90.000,C 0.000} C_DIS
LIN {X -73.517,Y -25.863,Z -41.115,A -90.000,B 90.000,C 0.000} C_DIS
LIN {X -73.389,Y -25.857,Z -41.137,A -90.000,B 90.000,C 0.000} C_DIS
LIN {X -72.609,Y -25.812,Z -41.236,A -90.000,B 90.000,C 0.000} C_DIS
LIN {X -72.149,Y -25.778,Z -41.298,A -90.000,B 90.000,C 0.000} C_DIS
LIN {X -71.983,Y -25.769,Z -41.327,A -90.000,B 90.000,C 0.000} C_DIS
LIN {X -71.803,Y -25.761,Z -41.364,A -90.000,B 90.000,C 0.000} C_DIS
LIN {X -71.713,Y -25.758,Z -41.384,A -90.000,B 90.000,C 0.000} C_DIS
LIN {X -71.375,Y -25.750,Z -41.469,A -90.000,B 90.000,C 0.000} C_DIS
LIN {X -71.196,Y -25.747,Z -41.520,A -90.000,B 90.000,C 0.000} C_DIS
LIN {X -71.020,Y -25.747,Z -41.578,A -90.000,B 90.000,C 0.000} C_DIS
LIN {X -70.049,Y -25.695,Z -41.815,A -90.000,B 90.000,C 0.000} C_DIS
LIN {X -69.861,Y -25.687,Z -41.866,A -90.000,B 90.000,C 0.000} C_DIS
LIN {X -69.724,Y -25.683,Z -41.905,A -90.000,B 90.000,C 0.000} C_DIS
LIN {X -69.443,Y -25.677,Z -41.997,A -90.000,B 90.000,C 0.000} C_DIS
LIN {X -69.299,Y -25.669,Z -42.031,A -90.000,B 90.000,C 0.000} C_DIS
LIN {X -68.852,Y -25.637,Z -42.142,A -90.000,B 90.000,C 0.000} C_DIS
LIN {X -68.579,Y -25.605,Z -42.182,A -90.000,B 90.000,C 0.000} C_DIS
LIN {X -68.395,Y -25.586,Z -42.216,A -90.000,B 90.000,C 0.000} C_DIS
LIN {X -66.895,Y -25.456,Z -42.551,A -90.000,B 90.000,C 0.000} C_DIS
LIN {X -66.393,Y -25.408,Z -42.657,A -90.000,B 90.000,C 0.000} C_DIS
LIN {X -65.960,Y -25.357,Z -42.723,A -90.000,B 90.000,C 0.000} C_DIS
LIN {X -65.844,Y -25.345,Z -42.744,A -90.000,B 90.000,C 0.000} C_DIS
LIN {X -65.579,Y -25.319,Z -42.797,A -90.000,B 90.000,C 0.000} C_DIS
LIN {X -65.459,Y -25.308,Z -42.826,A -90.000,B 90.000,C 0.000} C_DIS
LIN {X -65.459,Y -60.000,Z -42.826,A -90.000,B 90.000,C 0.000} C_DIS
LIN {X -87.599,Y -60.000,Z -40.529,A -90.000,B 90.000,C 0.000} C_DIS
LIN {X -87.599,Y -25.308,Z -40.529,A -90.000,B 90.000,C 0.000} C_DIS
LIN {X -87.278,Y -25.399,Z -40.580,A -90.000,B 90.000,C 0.000} C_DIS
LIN {X -87.115,Y -25.443,Z -40.609,A -90.000,B 90.000,C 0.000} C_DIS
LIN {X -86.723,Y -25.540,Z -40.682,A -90.000,B 90.000,C 0.000} C_DIS
LIN {X -86.466,Y -25.604,Z -40.739,A -90.000,B 90.000,C 0.000} C_DIS
LIN {X -86.286,Y -25.649,Z -40.783,A -90.000,B 90.000,C 0.000} C_DIS
LIN {X -85.795,Y -25.775,Z -40.922,A -90.000,B 90.000,C 0.000} C_DIS
LIN {X -85.551,Y -25.840,Z -41.001,A -90.000,B 90.000,C 0.000} C_DIS
LIN {X -85.155,Y -25.946,Z -41.136,A -90.000,B 90.000,C 0.000} C_DIS
LIN {X -84.937,Y -25.992,Z -41.211,A -90.000,B 90.000,C 0.000} C_DIS
LIN {X -84.538,Y -26.077,Z -41.359,A -90.000,B 90.000,C 0.000} C_DIS
LIN {X -84.093,Y -26.171,Z -41.532,A -90.000,B 90.000,C 0.000} C_DIS
LIN {X -83.571,Y -26.283,Z -41.750,A -90.000,B 90.000,C 0.000} C_DIS
LIN {X -83.115,Y -26.380,Z -41.954,A -90.000,B 90.000,C 0.000} C_DIS
LIN {X -83.035,Y -26.397,Z -41.991,A -90.000,B 90.000,C 0.000} C_DIS
LIN {X -82.880,Y -26.426,Z -42.031,A -90.000,B 90.000,C 0.000} C_DIS
LIN {X -82.742,Y -26.444,Z -42.068,A -90.000,B 90.000,C 0.000} C_DIS
LIN {X -82.450,Y -26.484,Z -42.156,A -90.000,B 90.000,C 0.000} C_DIS
LIN {X -81.907,Y -26.556,Z -42.336,A -90.000,B 90.000,C 0.000} C_DIS
LIN {X -81.716,Y -26.546,Z -42.101,A -90.000,B 90.000,C 0.000} C_DIS
LIN {X -81.601,Y -26.535,Z -41.967,A -90.000,B 90.000,C 0.000} C_DIS
LIN {X -81.411,Y -26.513,Z -41.761,A -90.000,B 90.000,C 0.000} C_DIS
LIN {X -81.316,Y -26.504,Z -41.665,A -90.000,B 90.000,C 0.000} C_DIS
LIN {X -81.192,Y -26.486,Z -41.544,A -90.000,B 90.000,C 0.000} C_DIS
LIN {X -81.026,Y -26.459,Z -41.388,A -90.000,B 90.000,C 0.000} C_DIS
LIN {X -80.885,Y -26.438,Z -41.265,A -90.000,B 90.000,C 0.000} C_DIS
LIN {X -80.786,Y -26.424,Z -41.182,A -90.000,B 90.000,C 0.000} C_DIS
LIN {X -80.643,Y -26.397,Z -41.065,A -90.000,B 90.000,C 0.000} C_DIS
LIN {X -80.381,Y -26.351,Z -40.870,A -90.000,B 90.000,C 0.000} C_DIS
LIN {X -80.236,Y -26.320,Z -40.769,A -90.000,B 90.000,C 0.000} C_DIS
LIN {X -80.135,Y -26.297,Z -40.701,A -90.000,B 90.000,C 0.000} C_DIS
LIN {X -79.847,Y -26.235,Z -40.522,A -90.000,B 90.000,C 0.000} C_DIS
LIN {X -79.780,Y -26.222,Z -40.484,A -90.000,B 90.000,C 0.000} C_DIS
LIN {X -79.625,Y -26.190,Z -40.397,A -90.000,B 90.000,C 0.000} C_DIS
LIN {X -79.509,Y -26.164,Z -40.335,A -90.000,B 90.000,C 0.000} C_DIS
LIN {X -79.316,Y -26.124,Z -40.237,A -90.000,B 90.000,C 0.000} C_DIS
LIN {X -79.138,Y -26.084,Z -40.153,A -90.000,B 90.000,C 0.000} C_DIS
LIN {X -78.843,Y -26.023,Z -40.027,A -90.000,B 90.000,C 0.000} C_DIS
LIN {X -78.488,Y -25.943,Z -39.893,A -90.000,B 90.000,C 0.000} C_DIS
LIN {X -78.237,Y -25.887,Z -39.810,A -90.000,B 90.000,C 0.000} C_DIS
LIN {X -77.390,Y -25.695,Z -39.556,A -90.000,B 90.000,C 0.000} C_DIS
LIN {X -77.080,Y -25.627,Z -39.472,A -90.000,B 90.000,C 0.000} C_DIS
LIN {X -76.954,Y -25.600,Z -39.441,A -90.000,B 90.000,C 0.000} C_DIS
LIN {X -76.755,Y -25.557,Z -39.397,A -90.000,B 90.000,C 0.000} C_DIS
LIN {X -76.273,Y -25.457,Z -39.306,A -90.000,B 90.000,C 0.000} C_DIS
LIN {X -76.028,Y -25.409,Z -39.267,A -90.000,B 90.000,C 0.000} C_DIS
LIN {X -75.653,Y -25.342,Z -39.219,A -90.000,B 90.000,C 0.000} C_DIS
LIN {X -75.521,Y -25.319,Z -39.207,A -90.000,B 90.000,C 0.000} C_DIS
LIN {X -75.444,Y -25.308,Z -39.201,A -90.000,B 90.000,C 0.000} C_DIS
LIN {X -75.444,Y -60.000,Z -39.201,A -90.000,B 90.000,C 0.000} C_DIS
LIN {X -85.655,Y -60.000,Z -38.916,A -90.000,B 90.000,C 0.000} C_DIS
LIN {X -85.655,Y -25.308,Z -38.916,A -90.000,B 90.000,C 0.000} C_DIS
LIN {X -85.258,Y -25.422,Z -39.027,A -90.000,B 90.000,C 0.000} C_DIS
LIN {X -85.114,Y -25.458,Z -39.069,A -90.000,B 90.000,C 0.000} C_DIS
LIN {X -84.981,Y -25.493,Z -39.112,A -90.000,B 90.000,C 0.000} C_DIS
LIN {X -84.837,Y -25.525,Z -39.159,A -90.000,B 90.000,C 0.000} C_DIS
LIN {X -84.191,Y -25.674,Z -39.383,A -90.000,B 90.000,C 0.000} C_DIS
LIN {X -83.768,Y -25.774,Z -39.538,A -90.000,B 90.000,C 0.000} C_DIS
LIN {X -83.279,Y -25.893,Z -39.726,A -90.000,B 90.000,C 0.000} C_DIS
LIN {X -83.095,Y -25.940,Z -39.802,A -90.000,B 90.000,C 0.000} C_DIS
LIN {X -82.820,Y -26.000,Z -39.917,A -90.000,B 90.000,C 0.000} C_DIS
LIN {X -82.715,Y -26.018,Z -39.962,A -90.000,B 90.000,C 0.000} C_DIS
LIN {X -82.479,Y -26.059,Z -40.069,A -90.000,B 90.000,C 0.000} C_DIS
LIN {X -82.348,Y -26.029,Z -39.950,A -90.000,B 90.000,C 0.000} C_DIS
LIN {X -82.175,Y -25.989,Z -39.804,A -90.000,B 90.000,C 0.000} C_DIS
LIN {X -81.866,Y -25.920,Z -39.556,A -90.000,B 90.000,C 0.000} C_DIS
LIN {X -81.560,Y -25.855,Z -39.333,A -90.000,B 90.000,C 0.000} C_DIS
LIN {X -81.345,Y -25.812,Z -39.183,A -90.000,B 90.000,C 0.000} C_DIS
LIN {X -81.197,Y -25.776,Z -39.088,A -90.000,B 90.000,C 0.000} C_DIS
LIN {X -80.955,Y -25.722,Z -38.939,A -90.000,B 90.000,C 0.000} C_DIS
LIN {X -80.826,Y -25.689,Z -38.865,A -90.000,B 90.000,C 0.000} C_DIS
LIN {X -80.680,Y -25.652,Z -38.785,A -90.000,B 90.000,C 0.000} C_DIS
LIN {X -80.474,Y -25.596,Z -38.677,A -90.000,B 90.000,C 0.000} C_DIS
LIN {X -80.164,Y -25.517,Z -38.528,A -90.000,B 90.000,C 0.000} C_DIS
LIN {X -79.994,Y -25.475,Z -38.452,A -90.000,B 90.000,C 0.000} C_DIS
LIN {X -79.633,Y -25.391,Z -38.301,A -90.000,B 90.000,C 0.000} C_DIS
LIN {X -79.249,Y -25.308,Z -38.156,A -90.000,B 90.000,C 0.000} C_DIS
LIN {X -79.249,Y -60.000,Z -38.156,A -90.000,B 90.000,C 0.000} C_DIS
LIN {X -97.773,Y -60.000,Z -53.012,A -90.000,B 90.000,C 0.000} C_DIS
LIN {X -97.773,Y -25.308,Z -53.012,A -90.000,B 90.000,C 0.000} C_DIS
LIN {X -97.993,Y -25.414,Z -52.525,A -90.000,B 90.000,C 0.000} C_DIS
LIN {X -98.035,Y -25.437,Z -52.426,A -90.000,B 90.000,C 0.000} C_DIS
LIN {X -98.085,Y -25.468,Z -52.286,A -90.000,B 90.000,C 0.000} C_DIS
LIN {X -98.116,Y -25.488,Z -52.197,A -90.000,B 90.000,C 0.000} C_DIS
LIN {X -98.174,Y -25.534,Z -51.990,A -90.000,B 90.000,C 0.000} C_DIS
LIN {X -98.253,Y -25.608,Z -51.666,A -90.000,B 90.000,C 0.000} C_DIS
LIN {X -98.322,Y -25.682,Z -51.349,A -90.000,B 90.000,C 0.000} C_DIS
LIN {X -98.356,Y -25.713,Z -51.172,A -90.000,B 90.000,C 0.000} C_DIS
LIN {X -98.367,Y -25.725,Z -51.107,A -90.000,B 90.000,C 0.000} C_DIS
LIN {X -98.390,Y -25.757,Z -50.932,A -90.000,B 90.000,C 0.000} C_DIS
LIN {X -98.405,Y -25.792,Z -50.757,A -90.000,B 90.000,C 0.000} C_DIS
LIN {X -98.413,Y -25.813,Z -50.645,A -90.000,B 90.000,C 0.000} C_DIS
LIN {X -98.427,Y -25.858,Z -50.373,A -90.000,B 90.000,C 0.000} C_DIS
LIN {X -98.428,Y -25.891,Z -50.174,A -90.000,B 90.000,C 0.000} C_DIS
LIN {X -98.417,Y -25.931,Z -49.890,A -90.000,B 90.000,C 0.000} C_DIS
LIN {X -98.400,Y -25.965,Z -49.663,A -90.000,B 90.000,C 0.000} C_DIS
LIN {X -98.390,Y -25.981,Z -49.568,A -90.000,B 90.000,C 0.000} C_DIS
LIN {X -98.371,Y -25.993,Z -49.423,A -90.000,B 90.000,C 0.000} C_DIS
LIN {X -98.353,Y -26.005,Z -49.274,A -90.000,B 90.000,C 0.000} C_DIS
LIN {X -98.340,Y -26.013,Z -49.190,A -90.000,B 90.000,C 0.000} C_DIS
LIN {X -98.317,Y -26.026,Z -49.059,A -90.000,B 90.000,C 0.000} C_DIS
LIN {X -98.288,Y -26.041,Z -48.925,A -90.000,B 90.000,C 0.000} C_DIS
LIN {X -98.251,Y -26.053,Z -48.778,A -90.000,B 90.000,C 0.000} C_DIS
LIN {X -98.190,Y -26.074,Z -48.554,A -90.000,B 90.000,C 0.000} C_DIS
LIN {X -98.132,Y -26.083,Z -48.373,A -90.000,B 90.000,C 0.000} C_DIS
LIN {X -98.074,Y -26.095,Z -48.216,A -90.000,B 90.000,C 0.000} C_DIS
LIN {X -98.017,Y -26.105,Z -48.080,A -90.000,B 90.000,C 0.000} C_DIS
LIN {X -97.968,Y -26.114,Z -47.972,A -90.000,B 90.000,C 0.000} C_DIS
LIN {X -97.934,Y -26.116,Z -47.901,A -90.000,B 90.000,C 0.000} C_DIS
LIN {X -97.891,Y -26.116,Z -47.801,A -90.000,B 90.000,C 0.000} C_DIS
LIN {X -97.835,Y -26.117,Z -47.680,A -90.000,B 90.000,C 0.000} C_DIS
LIN {X -97.719,Y -26.124,Z -47.458,A -90.000,B 90.000,C 0.000} C_DIS
LIN {X -97.685,Y -26.126,Z -47.393,A -90.000,B 90.000,C 0.000} C_DIS
LIN {X -97.601,Y -26.122,Z -47.244,A -90.000,B 90.000,C 0.000} C_DIS
LIN {X -97.531,Y -26.120,Z -47.130,A -90.000,B 90.000,C 0.000} C_DIS
LIN {X -97.455,Y -26.117,Z -47.014,A -90.000,B 90.000,C 0.000} C_DIS
LIN {X -97.325,Y -26.115,Z -46.833,A -90.000,B 90.000,C 0.000} C_DIS
LIN {X -97.194,Y -26.111,Z -46.676,A -90.000,B 90.000,C 0.000} C_DIS
LIN {X -97.146,Y -26.110,Z -46.620,A -90.000,B 90.000,C 0.000} C_DIS
LIN {X -97.071,Y -26.102,Z -46.536,A -90.000,B 90.000,C 0.000} C_DIS
LIN {X -96.958,Y -26.088,Z -46.402,A -90.000,B 90.000,C 0.000} C_DIS
LIN {X -96.718,Y -26.065,Z -46.138,A -90.000,B 90.000,C 0.000} C_DIS
LIN {X -96.689,Y -26.061,Z -46.107,A -90.000,B 90.000,C 0.000} C_DIS
LIN {X -96.523,Y -26.036,Z -45.951,A -90.000,B 90.000,C 0.000} C_DIS
LIN {X -96.410,Y -26.017,Z -45.854,A -90.000,B 90.000,C 0.000} C_DIS
LIN {X -96.288,Y -25.999,Z -45.758,A -90.000,B 90.000,C 0.000} C_DIS
LIN {X -96.177,Y -25.987,Z -45.676,A -90.000,B 90.000,C 0.000} C_DIS
LIN {X -96.037,Y -25.972,Z -45.578,A -90.000,B 90.000,C 0.000} C_DIS
LIN {X -95.833,Y -25.942,Z -45.419,A -90.000,B 90.000,C 0.000} C_DIS
LIN {X -95.633,Y -25.900,Z -45.283,A -90.000,B 90.000,C 0.000} C_DIS
LIN {X -95.379,Y -25.839,Z -45.124,A -90.000,B 90.000,C 0.000} C_DIS
LIN {X -95.272,Y -25.817,Z -45.061,A -90.000,B 90.000,C 0.000} C_DIS
LIN {X -95.121,Y -25.787,Z -44.980,A -90.000,B 90.000,C 0.000} C_DIS
LIN {X -94.989,Y -25.763,Z -44.916,A -90.000,B 90.000,C 0.000} C_DIS
LIN {X -94.831,Y -25.737,Z -44.845,A -90.000,B 90.000,C 0.000} C_DIS
LIN {X -94.606,Y -25.691,Z -44.754,A -90.000,B 90.000,C 0.000} C_DIS
LIN {X -94.447,Y -25.654,Z -44.700,A -90.000,B 90.000,C 0.000} C_DIS
LIN {X -94.308,Y -25.623,Z -44.655,A -90.000,B 90.000,C 0.000} C_DIS
LIN {X -94.178,Y -25.597,Z -44.619,A -90.000,B 90.000,C 0.000} C_DIS
LIN {X -94.116,Y -25.586,Z -44.603,A -90.000,B 90.000,C 0.000} C_DIS
LIN {X -93.962,Y -25.549,Z -44.553,A -90.000,B 90.000,C 0.000} C_DIS
LIN {X -93.752,Y -25.502,Z -44.493,A -90.000,B 90.000,C 0.000} C_DIS
LIN {X -93.606,Y -25.474,Z -44.457,A -90.000,B 90.000,C 0.000} C_DIS
LIN {X -93.354,Y -25.427,Z -44.407,A -90.000,B 90.000,C 0.000} C_DIS
LIN {X -93.203,Y -25.391,Z -44.383,A -90.000,B 90.000,C 0.000} C_DIS
LIN {X -93.106,Y -25.367,Z -44.369,A -90.000,B 90.000,C 0.000} C_DIS
LIN {X -92.849,Y -25.308,Z -44.345,A -90.000,B 90.000,C 0.000} C_DIS
LIN {X -92.757,Y -25.295,Z -44.337,A -90.000,B 90.000,C 0.000} C_DIS
LIN {X -92.497,Y -25.227,Z -44.319,A -90.000,B 90.000,C 0.000} C_DIS
LIN {X -92.334,Y -25.186,Z -44.314,A -90.000,B 90.000,C 0.000} C_DIS
LIN {X -92.180,Y -25.151,Z -44.313,A -90.000,B 90.000,C 0.000} C_DIS
LIN {X -91.965,Y -25.110,Z -44.319,A -90.000,B 90.000,C 0.000} C_DIS
LIN {X -91.770,Y -25.079,Z -44.335,A -90.000,B 90.000,C 0.000} C_DIS
LIN {X -91.593,Y -25.058,Z -44.361,A -90.000,B 90.000,C 0.000} C_DIS
LIN {X -91.485,Y -25.052,Z -44.383,A -90.000,B 90.000,C 0.000} C_DIS
LIN {X -91.434,Y -25.051,Z -44.396,A -90.000,B 90.000,C 0.000} C_DIS
LIN {X -91.338,Y -25.054,Z -44.423,A -90.000,B 90.000,C 0.000} C_DIS
LIN {X -91.249,Y -25.062,Z -44.455,A -90.000,B 90.000,C 0.000} C_DIS
LIN {X -91.208,Y -25.068,Z -44.472,A -90.000,B 90.000,C 0.000} C_DIS
LIN {X -91.131,Y -25.085,Z -44.509,A -90.000,B 90.000,C 0.000} C_DIS
LIN {X -91.095,Y -25.095,Z -44.529,A -90.000,B 90.000,C 0.000} C_DIS
LIN {X -91.029,Y -25.120,Z -44.572,A -90.000,B 90.000,C 0.000} C_DIS
LIN {X -90.999,Y -25.134,Z -44.594,A -90.000,B 90.000,C 0.000} C_DIS
LIN {X -90.944,Y -25.166,Z -44.642,A -90.000,B 90.000,C 0.000} C_DIS
LIN {X -90.896,Y -25.203,Z -44.692,A -90.000,B 90.000,C 0.000} C_DIS
LIN {X -90.875,Y -25.223,Z -44.719,A -90.000,B 90.000,C 0.000} C_DIS
LIN {X -90.837,Y -25.268,Z -44.774,A -90.000,B 90.000,C 0.000} C_DIS
LIN {X -90.821,Y -25.292,Z -44.803,A -90.000,B 90.000,C 0.000} C_DIS
LIN {X -90.794,Y -25.343,Z -44.863,A -90.000,B 90.000,C 0.000} C_DIS
LIN {X -90.764,Y -25.428,Z -44.958,A -90.000,B 90.000,C 0.000} C_DIS
LIN {X -90.750,Y -25.523,Z -45.059,A -90.000,B 90.000,C 0.000} C_DIS
LIN {X -90.748,Y -25.591,Z -45.130,A -90.000,B 90.000,C 0.000} C_DIS
LIN {X -90.752,Y -25.664,Z -45.203,A -90.000,B 90.000,C 0.000} C_DIS
LIN {X -90.762,Y -25.738,Z -45.279,A -90.000,B 90.000,C 0.000} C_DIS
LIN {X -90.777,Y -25.814,Z -45.356,A -90.000,B 90.000,C 0.000} C_DIS
LIN {X -90.812,Y -25.930,Z -45.477,A -90.000,B 90.000,C 0.000} C_DIS
LIN {X -90.858,Y -26.044,Z -45.603,A -90.000,B 90.000,C 0.000} C_DIS
LIN {X -90.917,Y -26.157,Z -45.732,A -90.000,B 90.000,C 0.000} C_DIS
LIN {X -90.962,Y -26.229,Z -45.821,A -90.000,B 90.000,C 0.000} C_DIS
LIN {X -91.012,Y -26.300,Z -45.911,A -90.000,B 90.000,C 0.000} C_DIS
LIN {X -91.127,Y -26.441,Z -46.097,A -90.000,B 90.000,C 0.000} C_DIS
LIN {X -91.261,Y -26.586,Z -46.288,A -90.000,B 90.000,C 0.000} C_DIS
LIN {X -91.334,Y -26.657,Z -46.385,A -90.000,B 90.000,C 0.000} C_DIS
LIN {X -91.412,Y -26.725,Z -46.483,A -90.000,B 90.000,C 0.000} C_DIS
LIN {X -91.494,Y -26.788,Z -46.583,A -90.000,B 90.000,C 0.000} C_DIS
LIN {X -91.579,Y -26.847,Z -46.683,A -90.000,B 90.000,C 0.000} C_DIS
LIN {X -91.669,Y -26.901,Z -46.784,A -90.000,B 90.000,C 0.000} C_DIS
LIN {X -91.762,Y -26.950,Z -46.886,A -90.000,B 90.000,C 0.000} C_DIS
LIN {X -91.859,Y -26.996,Z -46.988,A -90.000,B 90.000,C 0.000} C_DIS
LIN {X -92.063,Y -27.088,Z -47.194,A -90.000,B 90.000,C 0.000} C_DIS
LIN {X -92.170,Y -27.132,Z -47.298,A -90.000,B 90.000,C 0.000} C_DIS
LIN {X -92.280,Y -27.171,Z -47.402,A -90.000,B 90.000,C 0.000} C_DIS
LIN {X -92.393,Y -27.204,Z -47.506,A -90.000,B 90.000,C 0.000} C_DIS
LIN {X -92.509,Y -27.231,Z -47.610,A -90.000,B 90.000,C 0.000} C_DIS
LIN {X -92.628,Y -27.253,Z -47.714,A -90.000,B 90.000,C 0.000} C_DIS
LIN {X -92.749,Y -27.270,Z -47.818,A -90.000,B 90.000,C 0.000} C_DIS
LIN {X -92.998,Y -27.307,Z -48.025,A -90.000,B 90.000,C 0.000} C_DIS
LIN {X -93.126,Y -27.320,Z -48.128,A -90.000,B 90.000,C 0.000} C_DIS
LIN {X -93.257,Y -27.327,Z -48.230,A -90.000,B 90.000,C 0.000} C_DIS
LIN {X -93.389,Y -27.329,Z -48.332,A -90.000,B 90.000,C 0.000} C_DIS
LIN {X -93.523,Y -27.324,Z -48.433,A -90.000,B 90.000,C 0.000} C_DIS
LIN {X -93.796,Y -27.321,Z -48.632,A -90.000,B 90.000,C 0.000} C_DIS
LIN {X -93.935,Y -27.313,Z -48.730,A -90.000,B 90.000,C 0.000} C_DIS
LIN {X -94.359,Y -27.274,Z -49.018,A -90.000,B 90.000,C 0.000} C_DIS
LIN {X -94.502,Y -27.257,Z -49.111,A -90.000,B 90.000,C 0.000} C_DIS
LIN {X -94.791,Y -27.209,Z -49.293,A -90.000,B 90.000,C 0.000} C_DIS
LIN {X -95.083,Y -27.158,Z -49.468,A -90.000,B 90.000,C 0.000} C_DIS
LIN {X -95.229,Y -27.124,Z -49.553,A -90.000,B 90.000,C 0.000} C_DIS
LIN {X -95.375,Y -27.083,Z -49.636,A -90.000,B 90.000,C 0.000} C_DIS
LIN {X -95.669,Y -26.994,Z -49.795,A -90.000,B 90.000,C 0.000} C_DIS
LIN {X -95.815,Y -26.950,Z -49.872,A -90.000,B 90.000,C 0.000} C_DIS
LIN {X -95.961,Y -26.902,Z -49.946,A -90.000,B 90.000,C 0.000} C_DIS
LIN {X -96.106,Y -26.851,Z -50.018,A -90.000,B 90.000,C 0.000} C_DIS
LIN {X -96.252,Y -26.795,Z -50.087,A -90.000,B 90.000,C 0.000} C_DIS
LIN {X -96.539,Y -26.684,Z -50.217,A -90.000,B 90.000,C 0.000} C_DIS
LIN {X -96.682,Y -26.628,Z -50.278,A -90.000,B 90.000,C 0.000} C_DIS
LIN {X -96.824,Y -26.569,Z -50.336,A -90.000,B 90.000,C 0.000} C_DIS
LIN {X -96.964,Y -26.507,Z -50.391,A -90.000,B 90.000,C 0.000} C_DIS
LIN {X -97.241,Y -26.379,Z -50.491,A -90.000,B 90.000,C 0.000} C_DIS
LIN {X -97.377,Y -26.314,Z -50.537,A -90.000,B 90.000,C 0.000} C_DIS
LIN {X -97.644,Y -26.187,Z -50.617,A -90.000,B 90.000,C 0.000} C_DIS
LIN {X -97.774,Y -26.123,Z -50.652,A -90.000,B 90.000,C 0.000} C_DIS
LIN {X -98.029,Y -25.993,Z -50.711,A -90.000,B 90.000,C 0.000} C_DIS
LIN {X -98.275,Y -25.863,Z -50.754,A -90.000,B 90.000,C 0.000} C_DIS
LIN {X -98.394,Y -25.799,Z -50.769,A -90.000,B 90.000,C 0.000} C_DIS
LIN {X -98.510,Y -25.735,Z -50.781,A -90.000,B 90.000,C 0.000} C_DIS
LIN {X -98.624,Y -25.670,Z -50.788,A -90.000,B 90.000,C 0.000} C_DIS
LIN {X -98.789,Y -25.577,Z -50.790,A -90.000,B 90.000,C 0.000} C_DIS
LIN {X -98.895,Y -25.518,Z -50.786,A -90.000,B 90.000,C 0.000} C_DIS
LIN {X -98.997,Y -25.461,Z -50.778,A -90.000,B 90.000,C 0.000} C_DIS
LIN {X -99.096,Y -25.407,Z -50.765,A -90.000,B 90.000,C 0.000} C_DIS
LIN {X -99.239,Y -25.332,Z -50.736,A -90.000,B 90.000,C 0.000} C_DIS
LIN {X -99.329,Y -25.286,Z -50.710,A -90.000,B 90.000,C 0.000} C_DIS
LIN {X -99.415,Y -25.244,Z -50.680,A -90.000,B 90.000,C 0.000} C_DIS
LIN {X -99.498,Y -25.205,Z -50.645,A -90.000,B 90.000,C 0.000} C_DIS
LIN {X -99.614,Y -25.154,Z -50.582,A -90.000,B 90.000,C 0.000} C_DIS
LIN {X -99.686,Y -25.126,Z -50.533,A -90.000,B 90.000,C 0.000} C_DIS
LIN {X -99.754,Y -25.101,Z -50.479,A -90.000,B 90.000,C 0.000} C_DIS
LIN {X -99.817,Y -25.080,Z -50.419,A -90.000,B 90.000,C 0.000} C_DIS
LIN {X -99.875,Y -25.064,Z -50.354,A -90.000,B 90.000,C 0.000} C_DIS
LIN {X -99.929,Y -25.052,Z -50.283,A -90.000,B 90.000,C 0.000} C_DIS
LIN {X -99.978,Y -25.044,Z -50.206,A -90.000,B 90.000,C 0.000} C_DIS
LIN {X -100.022,Y -25.041,Z -50.123,A -90.000,B 90.000,C 0.000} C_DIS
LIN {X -100.060,Y -25.042,Z -50.034,A -90.000,B 90.000,C 0.000} C_DIS
LIN {X -100.094,Y -25.047,Z -49.939,A -90.000,B 90.000,C 0.000} C_DIS
LIN {X -100.134,Y -25.063,Z -49.785,A -90.000,B 90.000,C 0.000} C_DIS
LIN {X -100.153,Y -25.078,Z -49.674,A -90.000,B 90.000,C 0.000} C_DIS
LIN {X -100.167,Y -25.095,Z -49.557,A -90.000,B 90.000,C 0.000} C_DIS
LIN {X -100.175,Y -25.114,Z -49.433,A -90.000,B 90.000,C 0.000} C_DIS
LIN {X -100.177,Y -25.137,Z -49.303,A -90.000,B 90.000,C 0.000} C_DIS
LIN {X -100.173,Y -25.161,Z -49.166,A -90.000,B 90.000,C 0.000} C_DIS
LIN {X -100.163,Y -25.185,Z -49.022,A -90.000,B 90.000,C 0.000} C_DIS
LIN {X -100.147,Y -25.209,Z -48.871,A -90.000,B 90.000,C 0.000} C_DIS
LIN {X -100.124,Y -25.238,Z -48.714,A -90.000,B 90.000,C 0.000} C_DIS
LIN {X -100.077,Y -25.278,Z -48.463,A -90.000,B 90.000,C 0.000} C_DIS
LIN {X -100.037,Y -25.301,Z -48.288,A -90.000,B 90.000,C 0.000} C_DIS
LIN {X -100.014,Y -25.308,Z -48.197,A -90.000,B 90.000,C 0.000} C_DIS
LIN {X -99.961,Y -25.337,Z -47.987,A -90.000,B 90.000,C 0.000} C_DIS
LIN {X -99.881,Y -25.365,Z -47.721,A -90.000,B 90.000,C 0.000} C_DIS
LIN {X -99.843,Y -25.378,Z -47.611,A -90.000,B 90.000,C 0.000} C_DIS
LIN {X -99.783,Y -25.390,Z -47.454,A -90.000,B 90.000,C 0.000} C_DIS
LIN {X -99.702,Y -25.406,Z -47.259,A -90.000,B 90.000,C 0.000} C_DIS
LIN {X -99.639,Y -25.418,Z -47.122,A -90.000,B 90.000,C 0.000} C_DIS
LIN {X -99.607,Y -25.424,Z -47.042,A -90.000,B 90.000,C 0.000} C_DIS
LIN {X -99.510,Y -25.427,Z -46.832,A -90.000,B 90.000,C 0.000} C_DIS
LIN {X -99.319,Y -25.435,Z -46.470,A -90.000,B 90.000,C 0.000} C_DIS
LIN {X -99.216,Y -25.431,Z -46.290,A -90.000,B 90.000,C 0.000} C_DIS
LIN {X -99.156,Y -25.428,Z -46.191,A -90.000,B 90.000,C 0.000} C_DIS
LIN {X -99.022,Y -25.418,Z -45.986,A -90.000,B 90.000,C 0.000} C_DIS
LIN {X -98.969,Y -25.417,Z -45.910,A -90.000,B 90.000,C 0.000} C_DIS
LIN {X -98.804,Y -25.406,Z -45.689,A -90.000,B 90.000,C 0.000} C_DIS
LIN {X -98.585,Y -25.385,Z -45.435,A -90.000,B 90.000,C 0.000} C_DIS
LIN {X -98.516,Y -25.379,Z -45.357,A -90.000,B 90.000,C 0.000} C_DIS
LIN {X -98.367,Y -25.359,Z -45.185,A -90.000,B 90.000,C 0.000} C_DIS
LIN {X -98.297,Y -25.351,Z -45.108,A -90.000,B 90.000,C 0.000} C_DIS
LIN {X -98.084,Y -25.314,Z -44.883,A -90.000,B 90.000,C 0.000} C_DIS
LIN {X -98.053,Y -25.308,Z -44.853,A -90.000,B 90.000,C 0.000} C_DIS
LIN {X -98.053,Y -60.000,Z -44.853,A -90.000,B 90.000,C 0.000} C_DIS
LIN {X -87.848,Y -60.000,Z -65.271,A -90.000,B 90.000,C 0.000} C_DIS
LIN {X -87.848,Y -25.308,Z -65.271,A -90.000,B 90.000,C 0.000} C_DIS
LIN {X -87.954,Y -25.364,Z -65.059,A -90.000,B 90.000,C 0.000} C_DIS
LIN {X -88.145,Y -25.482,Z -64.654,A -90.000,B 90.000,C 0.000} C_DIS
LIN {X -88.249,Y -25.499,Z -64.544,A -90.000,B 90.000,C 0.000} C_DIS
LIN {X -88.441,Y -25.518,Z -64.366,A -90.000,B 90.000,C 0.000} C_DIS
LIN {X -88.866,Y -25.555,Z -63.970,A -90.000,B 90.000,C 0.000} C_DIS
LIN {X -89.179,Y -25.575,Z -63.690,A -90.000,B 90.000,C 0.000} C_DIS
LIN {X -90.085,Y -25.626,Z -62.873,A -90.000,B 90.000,C 0.000} C_DIS
LIN {X -90.537,Y -25.641,Z -62.472,A -90.000,B 90.000,C 0.000} C_DIS
LIN {X -91.018,Y -25.658,Z -62.042,A -90.000,B 90.000,C 0.000} C_DIS
LIN {X -91.550,Y -25.665,Z -61.554,A -90.000,B 90.000,C 0.000} C_DIS
LIN {X -91.931,Y -25.674,Z -61.191,A -90.000,B 90.000,C 0.000} C_DIS
LIN {X -92.112,Y -25.679,Z -61.014,A -90.000,B 90.000,C 0.000} C_DIS
LIN {X -92.388,Y -25.675,Z -60.740,A -90.000,B 90.000,C 0.000} C_DIS
LIN {X -92.907,Y -25.661,Z -60.215,A -90.000,B 90.000,C 0.000} C_DIS
LIN {X -93.107,Y -25.651,Z -60.010,A -90.000,B 90.000,C 0.000} C_DIS
LIN {X -93.379,Y -25.633,Z -59.722,A -90.000,B 90.000,C 0.000} C_DIS
LIN {X -93.553,Y -25.623,Z -59.535,A -90.000,B 90.000,C 0.000} C_DIS
LIN {X -93.817,Y -25.609,Z -59.245,A -90.000,B 90.000,C 0.000} C_DIS
LIN {X -93.958,Y -25.596,Z -59.085,A -90.000,B 90.000,C 0.000} C_DIS
LIN {X -94.042,Y -25.589,Z -58.985,A -90.000,B 90.000,C 0.000} C_DIS
LIN {X -94.458,Y -25.564,Z -58.491,A -90.000,B 90.000,C 0.000} C_DIS
LIN {X -94.693,Y -25.542,Z -58.184,A -90.000,B 90.000,C 0.000} C_DIS
LIN {X -94.944,Y -25.514,Z -57.851,A -90.000,B 90.000,C 0.000} C_DIS
LIN {X -94.986,Y -25.512,Z -57.795,A -90.000,B 90.000,C 0.000} C_DIS
LIN {X -95.279,Y -25.479,Z -57.462,A -90.000,B 90.000,C 0.000} C_DIS
LIN {X -95.521,Y -25.453,Z -57.161,A -90.000,B 90.000,C 0.000} C_DIS
LIN {X -95.944,Y -25.405,Z -56.607,A -90.000,B 90.000,C 0.000} C_DIS
LIN {X -96.033,Y -25.393,Z -56.485,A -90.000,B 90.000,C 0.000} C_DIS
LIN {X -96.284,Y -25.350,Z -56.130,A -90.000,B 90.000,C 0.000} C_DIS
LIN {X -96.354,Y -25.336,Z -56.021,A -90.000,B 90.000,C 0.000} C_DIS
LIN {X -96.475,Y -25.312,Z -55.820,A -90.000,B 90.000,C 0.000} C_DIS
LIN {X -96.492,Y -25.308,Z -55.789,A -90.000,B 90.000,C 0.000} C_DIS
LIN {X -96.492,Y -60.000,Z -55.789,A -90.000,B 90.000,C 0.000} C_DIS
LIN {X -104.903,Y -60.000,Z -243.561,A -90.000,B 90.000,C 0.000} C_DIS
LIN {X -104.903,Y -25.308,Z -243.561,A -90.000,B 90.000,C 0.000} C_DIS
LIN {X -102.194,Y -25.308,Z -241.677,A -90.000,B 90.000,C 0.000} C_DIS
LIN {X -101.011,Y -25.308,Z -240.895,A -90.000,B 90.000,C 0.000} C_DIS
LIN {X -94.263,Y -25.308,Z -236.359,A -90.000,B 90.000,C 0.000} C_DIS
LIN {X -86.123,Y -25.308,Z -231.074,A -90.000,B 90.000,C 0.000} C_DIS
LIN {X -80.853,Y -25.308,Z -227.781,A -90.000,B 90.000,C 0.000} C_DIS
LIN {X -77.684,Y -25.308,Z -225.808,A -90.000,B 90.000,C 0.000} C_DIS
LIN {X -77.295,Y -25.308,Z -225.569,A -90.000,B 90.000,C 0.000} C_DIS
LIN {X -70.073,Y -25.308,Z -221.258,A -90.000,B 90.000,C 0.000} C_DIS
LIN {X -68.679,Y -25.308,Z -220.428,A -90.000,B 90.000,C 0.000} C_DIS
LIN {X -62.658,Y -25.308,Z -216.937,A -90.000,B 90.000,C 0.000} C_DIS
LIN {X -60.459,Y -25.308,Z -215.671,A -90.000,B 90.000,C 0.000} C_DIS
LIN {X -53.310,Y -25.308,Z -211.603,A -90.000,B 90.000,C 0.000} C_DIS
LIN {X -52.583,Y -25.308,Z -211.198,A -90.000,B 90.000,C 0.000} C_DIS
LIN {X -47.034,Y -25.308,Z -208.061,A -90.000,B 90.000,C 0.000} C_DIS
LIN {X -45.509,Y -25.308,Z -207.218,A -90.000,B 90.000,C 0.000} C_DIS
LIN {X -39.976,Y -25.308,Z -204.060,A -90.000,B 90.000,C 0.000} C_DIS
LIN {X -37.189,Y -25.308,Z -202.425,A -90.000,B 90.000,C 0.000} C_DIS
LIN {X -35.487,Y -25.308,Z -201.428,A -90.000,B 90.000,C 0.000} C_DIS
LIN {X -35.190,Y -25.308,Z -201.257,A -90.000,B 90.000,C 0.000} C_DIS
LIN {X -31.529,Y -25.308,Z -199.005,A -90.000,B 90.000,C 0.000} C_DIS
LIN {X -31.140,Y -25.308,Z -198.767,A -90.000,B 90.000,C 0.000} C_DIS
LIN {X -28.479,Y -25.308,Z -197.001,A -90.000,B 90.000,C 0.000} C_DIS
LIN {X -27.830,Y -25.308,Z -196.555,A -90.000,B 90.000,C 0.000} C_DIS
LIN {X -25.708,Y -25.308,Z -195.008,A -90.000,B 90.000,C 0.000} C_DIS
LIN {X -24.631,Y -25.308,Z -194.201,A -90.000,B 90.000,C 0.000} C_DIS
LIN {X -24.323,Y -25.308,Z -193.952,A -90.000,B 90.000,C 0.000} C_DIS
LIN {X -21.893,Y -25.308,Z -191.950,A -90.000,B 90.000,C 0.000} C_DIS
LIN {X -20.595,Y -25.308,Z -190.767,A -90.000,B 90.000,C 0.000} C_DIS
LIN {X -19.347,Y -25.308,Z -189.618,A -90.000,B 90.000,C 0.000} C_DIS
LIN {X -18.518,Y -25.308,Z -188.795,A -90.000,B 90.000,C 0.000} C_DIS
LIN {X -16.584,Y -25.308,Z -186.854,A -90.000,B 90.000,C 0.000} C_DIS
LIN {X -16.178,Y -25.308,Z -186.421,A -90.000,B 90.000,C 0.000} C_DIS
LIN {X -15.323,Y -25.308,Z -185.491,A -90.000,B 90.000,C 0.000} C_DIS
LIN {X -14.666,Y -25.308,Z -184.770,A -90.000,B 90.000,C 0.000} C_DIS
LIN {X -14.035,Y -25.308,Z -184.074,A -90.000,B 90.000,C 0.000} C_DIS
LIN {X -12.793,Y -25.308,Z -182.578,A -90.000,B 90.000,C 0.000} C_DIS
LIN {X -11.459,Y -25.308,Z -180.943,A -90.000,B 90.000,C 0.000} C_DIS
LIN {X -10.680,Y -25.308,Z -179.887,A -90.000,B 90.000,C 0.000} C_DIS
LIN {X -9.151,Y -25.308,Z -177.747,A -90.000,B 90.000,C 0.000} C_DIS
LIN {X -7.830,Y -25.308,Z -175.547,A -90.000,B 90.000,C 0.000} C_DIS
LIN {X -7.200,Y -25.308,Z -174.486,A -90.000,B 90.000,C 0.000} C_DIS
LIN {X -6.272,Y -25.308,Z -172.550,A -90.000,B 90.000,C 0.000} C_DIS
LIN {X -5.642,Y -25.308,Z -171.212,A -90.000,B 90.000,C 0.000} C_DIS
LIN {X -5.180,Y -25.308,Z -169.873,A -90.000,B 90.000,C 0.000} C_DIS
LIN {X -4.534,Y -25.308,Z -167.967,A -90.000,B 90.000,C 0.000} C_DIS
LIN {X -4.128,Y -25.308,Z -165.734,A -90.000,B 90.000,C 0.000} C_DIS
LIN {X -4.024,Y -25.308,Z -165.165,A -90.000,B 90.000,C 0.000} C_DIS
LIN {X -4.030,Y -25.308,Z -164.925,A -90.000,B 90.000,C 0.000} C_DIS
LIN {X -4.039,Y -25.308,Z -162.887,A -90.000,B 90.000,C 0.000} C_DIS
LIN {X -4.452,Y -25.308,Z -161.568,A -90.000,B 90.000,C 0.000} C_DIS
LIN {X -4.517,Y -25.308,Z -161.333,A -90.000,B 90.000,C 0.000} C_DIS
LIN {X -4.923,Y -25.308,Z -160.727,A -90.000,B 90.000,C 0.000} C_DIS
LIN {X -5.159,Y -25.308,Z -160.353,A -90.000,B 90.000,C 0.000} C_DIS
LIN {X -5.261,Y -25.308,Z -160.182,A -90.000,B 90.000,C 0.000} C_DIS
LIN {X -5.737,Y -25.308,Z -159.724,A -90.000,B 90.000,C 0.000} C_DIS
LIN {X -6.357,Y -25.308,Z -159.072,A -90.000,B 90.000,C 0.000} C_DIS
LIN {X -6.584,Y -25.308,Z -158.903,A -90.000,B 90.000,C 0.000} C_DIS
LIN {X -7.845,Y -25.308,Z -157.869,A -90.000,B 90.000,C 0.000} C_DIS
LIN {X -8.105,Y -25.308,Z -157.672,A -90.000,B 90.000,C 0.000} C_DIS
LIN {X -9.229,Y -25.308,Z -156.814,A -90.000,B 90.000,C 0.000} C_DIS
LIN {X -9.691,Y -25.308,Z -156.454,A -90.000,B 90.000,C 0.000} C_DIS
LIN {X -9.860,Y -25.308,Z -156.318,A -90.000,B 90.000,C 0.000} C_DIS
LIN {X -11.704,Y -25.308,Z -154.924,A -90.000,B 90.000,C 0.000} C_DIS
LIN {X -12.439,Y -25.308,Z -154.328,A -90.000,B 90.000,C 0.000} C_DIS
LIN {X -13.938,Y -25.308,Z -153.183,A -90.000,B 90.000,C 0.000} C_DIS
LIN {X -14.692,Y -25.308,Z -152.562,A -90.000,B 90.000,C 0.000} C_DIS
LIN {X -16.530,Y -25.308,Z -151.110,A -90.000,B 90.000,C 0.000} C_DIS
LIN {X -17.337,Y -25.308,Z -150.432,A -90.000,B 90.000,C 0.000} C_DIS
LIN {X -19.561,Y -25.308,Z -148.591,A -90.000,B 90.000,C 0.000} C_DIS
LIN {X -19.918,Y -25.308,Z -148.291,A -90.000,B 90.000,C 0.000} C_DIS
LIN {X -23.159,Y -25.308,Z -145.361,A -90.000,B 90.000,C 0.000} C_DIS
LIN {X -26.558,Y -25.308,Z -141.914,A -90.000,B 90.000,C 0.000} C_DIS
LIN {X -26.681,Y -25.308,Z -141.787,A -90.000,B 90.000,C 0.000} C_DIS
LIN {X -27.614,Y -25.308,Z -140.661,A -90.000,B 90.000,C 0.000} C_DIS
LIN {X -28.814,Y -25.308,Z -139.302,A -90.000,B 90.000,C 0.000} C_DIS
LIN {X -29.254,Y -25.308,Z -138.812,A -90.000,B 90.000,C 0.000} C_DIS
LIN {X -30.219,Y -25.308,Z -137.843,A -90.000,B 90.000,C 0.000} C_DIS
LIN {X -30.240,Y -25.308,Z -137.818,A -90.000,B 90.000,C 0.000} C_DIS
LIN {X -30.527,Y -25.308,Z -137.478,A -90.000,B 90.000,C 0.000} C_DIS
LIN {X -32.674,Y -25.308,Z -134.829,A -90.000,B 90.000,C 0.000} C_DIS
LIN {X -33.314,Y -25.308,Z -134.051,A -90.000,B 90.000,C 0.000} C_DIS
LIN {X -33.644,Y -25.308,Z -133.567,A -90.000,B 90.000,C 0.000} C_DIS
LIN {X -35.907,Y -25.308,Z -130.179,A -90.000,B 90.000,C 0.000} C_DIS
LIN {X -38.052,Y -25.308,Z -126.263,A -90.000,B 90.000,C 0.000} C_DIS
LIN {X -38.234,Y -25.308,Z -125.927,A -90.000,B 90.000,C 0.000} C_DIS
LIN {X -38.969,Y -25.308,Z -124.276,A -90.000,B 90.000,C 0.000} C_DIS
LIN {X -39.528,Y -25.308,Z -123.145,A -90.000,B 90.000,C 0.000} C_DIS
LIN {X -39.731,Y -25.308,Z -122.729,A -90.000,B 90.000,C 0.000} C_DIS
LIN {X -40.598,Y -25.308,Z -120.751,A -90.000,B 90.000,C 0.000} C_DIS
LIN {X -40.869,Y -25.308,Z -120.117,A -90.000,B 90.000,C 0.000} C_DIS
LIN {X -41.115,Y -25.308,Z -119.391,A -90.000,B 90.000,C 0.000} C_DIS
LIN {X -41.705,Y -25.308,Z -117.935,A -90.000,B 90.000,C 0.000} C_DIS
LIN {X -41.904,Y -25.308,Z -117.361,A -90.000,B 90.000,C 0.000} C_DIS
LIN {X -42.504,Y -25.308,Z -116.062,A -90.000,B 90.000,C 0.000} C_DIS
LIN {X -42.662,Y -25.308,Z -115.687,A -90.000,B 90.000,C 0.000} C_DIS
LIN {X -43.491,Y -25.308,Z -114.207,A -90.000,B 90.000,C 0.000} C_DIS
LIN {X -43.702,Y -25.308,Z -113.817,A -90.000,B 90.000,C 0.000} C_DIS
LIN {X -44.836,Y -25.308,Z -112.099,A -90.000,B 90.000,C 0.000} C_DIS
LIN {X -45.269,Y -25.308,Z -111.445,A -90.000,B 90.000,C 0.000} C_DIS
LIN {X -46.285,Y -25.308,Z -110.026,A -90.000,B 90.000,C 0.000} C_DIS
LIN {X -47.588,Y -25.308,Z -108.259,A -90.000,B 90.000,C 0.000} C_DIS
LIN {X -48.398,Y -25.308,Z -107.210,A -90.000,B 90.000,C 0.000} C_DIS
LIN {X -49.300,Y -25.308,Z -106.007,A -90.000,B 90.000,C 0.000} C_DIS
LIN {X -49.628,Y -25.308,Z -105.593,A -90.000,B 90.000,C 0.000} C_DIS
LIN {X -50.998,Y -25.308,Z -103.790,A -90.000,B 90.000,C 0.000} C_DIS
LIN {X -52.105,Y -25.308,Z -102.407,A -90.000,B 90.000,C 0.000} C_DIS
LIN {X -52.748,Y -25.308,Z -101.570,A -90.000,B 90.000,C 0.000} C_DIS
LIN {X -54.235,Y -25.308,Z -99.627,A -90.000,B 90.000,C 0.000} C_DIS
LIN {X -54.801,Y -25.308,Z -98.876,A -90.000,B 90.000,C 0.000} C_DIS
LIN {X -56.234,Y -25.308,Z -96.929,A -90.000,B 90.000,C 0.000} C_DIS
LIN {X -56.854,Y -25.308,Z -96.117,A -90.000,B 90.000,C 0.000} C_DIS
LIN {X -57.167,Y -25.308,Z -95.700,A -90.000,B 90.000,C 0.000} C_DIS
LIN {X -57.564,Y -25.308,Z -95.164,A -90.000,B 90.000,C 0.000} C_DIS
LIN {X -58.866,Y -25.308,Z -93.463,A -90.000,B 90.000,C 0.000} C_DIS
LIN {X -59.173,Y -25.308,Z -93.061,A -90.000,B 90.000,C 0.000} C_DIS
LIN {X -60.034,Y -25.308,Z -91.955,A -90.000,B 90.000,C 0.000} C_DIS
LIN {X -60.864,Y -25.308,Z -90.850,A -90.000,B 90.000,C 0.000} C_DIS
LIN {X -61.141,Y -25.308,Z -90.497,A -90.000,B 90.000,C 0.000} C_DIS
LIN {X -61.684,Y -25.308,Z -89.844,A -90.000,B 90.000,C 0.000} C_DIS
LIN {X -63.073,Y -25.308,Z -88.131,A -90.000,B 90.000,C 0.000} C_DIS
LIN {X -64.370,Y -25.308,Z -86.669,A -90.000,B 90.000,C 0.000} C_DIS
LIN {X -64.921,Y -25.308,Z -86.027,A -90.000,B 90.000,C 0.000} C_DIS
LIN {X -66.300,Y -25.308,Z -84.542,A -90.000,B 90.000,C 0.000} C_DIS
LIN {X -66.685,Y -25.308,Z -84.113,A -90.000,B 90.000,C 0.000} C_DIS
LIN {X -66.936,Y -25.308,Z -83.844,A -90.000,B 90.000,C 0.000} C_DIS
LIN {X -68.468,Y -25.308,Z -82.166,A -90.000,B 90.000,C 0.000} C_DIS
LIN {X -69.891,Y -25.308,Z -80.647,A -90.000,B 90.000,C 0.000} C_DIS
LIN {X -70.140,Y -25.308,Z -80.374,A -90.000,B 90.000,C 0.000} C_DIS
LIN {X -70.461,Y -25.308,Z -80.039,A -90.000,B 90.000,C 0.000} C_DIS
LIN {X -70.810,Y -25.308,Z -79.667,A -90.000,B 90.000,C 0.000} C_DIS
LIN {X -71.798,Y -25.308,Z -78.600,A -90.000,B 90.000,C 0.000} C_DIS
LIN {X -72.090,Y -25.308,Z -78.295,A -90.000,B 90.000,C 0.000} C_DIS
LIN {X -73.156,Y -25.308,Z -77.145,A -90.000,B 90.000,C 0.000} C_DIS
LIN {X -73.853,Y -25.308,Z -76.469,A -90.000,B 90.000,C 0.000} C_DIS
LIN {X -74.280,Y -25.308,Z -76.050,A -90.000,B 90.000,C 0.000} C_DIS
LIN {X -74.872,Y -25.308,Z -75.571,A -90.000,B 90.000,C 0.000} C_DIS
LIN {X -75.019,Y -25.308,Z -75.491,A -90.000,B 90.000,C 0.000} C_DIS
LIN {X -75.167,Y -25.308,Z -75.494,A -90.000,B 90.000,C 0.000} C_DIS
LIN {X -75.323,Y -25.308,Z -75.486,A -90.000,B 90.000,C 0.000} C_DIS
LIN {X -75.362,Y -25.308,Z -75.489,A -90.000,B 90.000,C 0.000} C_DIS
LIN {X -75.785,Y -25.308,Z -75.468,A -90.000,B 90.000,C 0.000} C_DIS
LIN {X -76.063,Y -25.308,Z -75.435,A -90.000,B 90.000,C 0.000} C_DIS
LIN {X -76.887,Y -25.308,Z -75.396,A -90.000,B 90.000,C 0.000} C_DIS
LIN {X -77.326,Y -25.308,Z -75.321,A -90.000,B 90.000,C 0.000} C_DIS
LIN {X -77.968,Y -25.308,Z -75.161,A -90.000,B 90.000,C 0.000} C_DIS
LIN {X -78.473,Y -25.308,Z -75.050,A -90.000,B 90.000,C 0.000} C_DIS
LIN {X -78.880,Y -25.308,Z -74.931,A -90.000,B 90.000,C 0.000} C_DIS
LIN {X -79.195,Y -25.308,Z -74.831,A -90.000,B 90.000,C 0.000} C_DIS
LIN {X -79.974,Y -25.308,Z -74.501,A -90.000,B 90.000,C 0.000} C_DIS
LIN {X -80.397,Y -25.308,Z -74.294,A -90.000,B 90.000,C 0.000} C_DIS
LIN {X -80.690,Y -25.308,Z -74.135,A -90.000,B 90.000,C 0.000} C_DIS
LIN {X -81.578,Y -25.308,Z -73.630,A -90.000,B 90.000,C 0.000} C_DIS
LIN {X -81.719,Y -25.308,Z -73.539,A -90.000,B 90.000,C 0.000} C_DIS
LIN {X -82.151,Y -25.308,Z -73.232,A -90.000,B 90.000,C 0.000} C_DIS
LIN {X -82.492,Y -25.308,Z -72.952,A -90.000,B 90.000,C 0.000} C_DIS
LIN {X -82.799,Y -25.308,Z -72.693,A -90.000,B 90.000,C 0.000} C_DIS
LIN {X -83.106,Y -25.308,Z -72.377,A -90.000,B 90.000,C 0.000} C_DIS
LIN {X -83.420,Y -25.308,Z -72.035,A -90.000,B 90.000,C 0.000} C_DIS
LIN {X -83.703,Y -25.308,Z -71.740,A -90.000,B 90.000,C 0.000} C_DIS
LIN {X -83.972,Y -25.308,Z -71.391,A -90.000,B 90.000,C 0.000} C_DIS
LIN {X -84.185,Y -25.308,Z -71.082,A -90.000,B 90.000,C 0.000} C_DIS
LIN {X -84.393,Y -25.308,Z -70.746,A -90.000,B 90.000,C 0.000} C_DIS
LIN {X -84.621,Y -25.308,Z -70.368,A -90.000,B 90.000,C 0.000} C_DIS
LIN {X -84.805,Y -25.308,Z -69.967,A -90.000,B 90.000,C 0.000} C_DIS
LIN {X -84.903,Y -25.308,Z -69.730,A -90.000,B 90.000,C 0.000} C_DIS
LIN {X -85.079,Y -25.308,Z -69.337,A -90.000,B 90.000,C 0.000} C_DIS
LIN {X -85.218,Y -25.308,Z -68.918,A -90.000,B 90.000,C 0.000} C_DIS
LIN {X -85.267,Y -25.308,Z -68.780,A -90.000,B 90.000,C 0.000} C_DIS
LIN {X -85.366,Y -25.308,Z -68.414,A -90.000,B 90.000,C 0.000} C_DIS
LIN {X -85.437,Y -25.308,Z -68.162,A -90.000,B 90.000,C 0.000} C_DIS
LIN {X -85.531,Y -25.308,Z -67.749,A -90.000,B 90.000,C 0.000} C_DIS
LIN {X -85.535,Y -25.308,Z -67.719,A -90.000,B 90.000,C 0.000} C_DIS
LIN {X -85.561,Y -25.308,Z -67.624,A -90.000,B 90.000,C 0.000} C_DIS
LIN {X -85.583,Y -25.308,Z -67.512,A -90.000,B 90.000,C 0.000} C_DIS
LIN {X -85.594,Y -25.308,Z -67.473,A -90.000,B 90.000,C 0.000} C_DIS
LIN {X -85.660,Y -25.308,Z -67.350,A -90.000,B 90.000,C 0.000} C_DIS
LIN {X -85.716,Y -25.308,Z -67.230,A -90.000,B 90.000,C 0.000} C_DIS
LIN {X -85.864,Y -25.308,Z -67.028,A -90.000,B 90.000,C 0.000} C_DIS
LIN {X -85.944,Y -25.308,Z -66.909,A -90.000,B 90.000,C 0.000} C_DIS
LIN {X -86.280,Y -25.308,Z -66.519,A -90.000,B 90.000,C 0.000} C_DIS
LIN {X -86.526,Y -25.308,Z -66.269,A -90.000,B 90.000,C 0.000} C_DIS
LIN {X -86.798,Y -25.308,Z -66.032,A -90.000,B 90.000,C 0.000} C_DIS
LIN {X -87.095,Y -25.308,Z -65.813,A -90.000,B 90.000,C 0.000} C_DIS
LIN {X -87.388,Y -25.308,Z -65.588,A -90.000,B 90.000,C 0.000} C_DIS
LIN {X -87.726,Y -25.308,Z -65.358,A -90.000,B 90.000,C 0.000} C_DIS
LIN {X -88.113,Y -25.308,Z -65.082,A -90.000,B 90.000,C 0.000} C_DIS
LIN {X -89.027,Y -25.308,Z -64.460,A -90.000,B 90.000,C 0.000} C_DIS
LIN {X -89.376,Y -25.308,Z -64.214,A -90.000,B 90.000,C 0.000} C_DIS
LIN {X -90.084,Y -25.308,Z -63.728,A -90.000,B 90.000,C 0.000} C_DIS
LIN {X -90.363,Y -25.308,Z -63.523,A -90.000,B 90.000,C 0.000} C_DIS
LIN {X -91.148,Y -25.308,Z -62.958,A -90.000,B 90.000,C 0.000} C_DIS
LIN {X -91.366,Y -25.308,Z -62.786,A -90.000,B 90.000,C 0.000} C_DIS
LIN {X -92.078,Y -25.308,Z -62.214,A -90.000,B 90.000,C 0.000} C_DIS
LIN {X -92.554,Y -25.308,Z -61.797,A -90.000,B 90.000,C 0.000} C_DIS
LIN {X -93.035,Y -25.308,Z -61.323,A -90.000,B 90.000,C 0.000} C_DIS
LIN {X -93.371,Y -25.308,Z -60.983,A -90.000,B 90.000,C 0.000} C_DIS
LIN {X -93.614,Y -25.308,Z -60.696,A -90.000,B 90.000,C 0.000} C_DIS
LIN {X -94.092,Y -25.308,Z -60.141,A -90.000,B 90.000,C 0.000} C_DIS
LIN {X -94.286,Y -25.308,Z -59.907,A -90.000,B 90.000,C 0.000} C_DIS
LIN {X -94.353,Y -25.308,Z -59.822,A -90.000,B 90.000,C 0.000} C_DIS
LIN {X -94.835,Y -25.308,Z -59.127,A -90.000,B 90.000,C 0.000} C_DIS
LIN {X -94.937,Y -25.308,Z -58.963,A -90.000,B 90.000,C 0.000} C_DIS
LIN {X -95.171,Y -25.308,Z -58.552,A -90.000,B 90.000,C 0.000} C_DIS
LIN {X -95.402,Y -25.308,Z -58.201,A -90.000,B 90.000,C 0.000} C_DIS
LIN {X -95.562,Y -25.308,Z -57.944,A -90.000,B 90.000,C 0.000} C_DIS
LIN {X -96.114,Y -25.308,Z -56.919,A -90.000,B 90.000,C 0.000} C_DIS
LIN {X -96.345,Y -25.308,Z -56.371,A -90.000,B 90.000,C 0.000} C_DIS
LIN {X -96.433,Y -25.308,Z -56.103,A -90.000,B 90.000,C 0.000} C_DIS
LIN {X -96.488,Y -25.308,Z -55.818,A -90.000,B 90.000,C 0.000} C_DIS
LIN {X -96.518,Y -25.308,Z -55.583,A -90.000,B 90.000,C 0.000} C_DIS
LIN {X -96.497,Y -25.308,Z -55.344,A -90.000,B 90.000,C 0.000} C_DIS
LIN {X -96.402,Y -25.308,Z -55.005,A -90.000,B 90.000,C 0.000} C_DIS
LIN {X -96.337,Y -25.308,Z -54.793,A -90.000,B 90.000,C 0.000} C_DIS
LIN {X -96.290,Y -25.308,Z -54.705,A -90.000,B 90.000,C 0.000} C_DIS
LIN {X -96.621,Y -25.308,Z -54.367,A -90.000,B 90.000,C 0.000} C_DIS
LIN {X -97.347,Y -25.308,Z -53.553,A -90.000,B 90.000,C 0.000} C_DIS
LIN {X -97.548,Y -25.308,Z -53.302,A -90.000,B 90.000,C 0.000} C_DIS
LIN {X -98.383,Y -25.308,Z -52.225,A -90.000,B 90.000,C 0.000} C_DIS
LIN {X -98.603,Y -25.308,Z -51.916,A -90.000,B 90.000,C 0.000} C_DIS
LIN {X -98.774,Y -25.308,Z -51.654,A -90.000,B 90.000,C 0.000} C_DIS
LIN {X -98.912,Y -25.308,Z -51.420,A -90.000,B 90.000,C 0.000} C_DIS
LIN {X -99.089,Y -25.308,Z -51.084,A -90.000,B 90.000,C 0.000} C_DIS
LIN {X -99.367,Y -25.308,Z -50.538,A -90.000,B 90.000,C 0.000} C_DIS
LIN {X -99.450,Y -25.308,Z -50.360,A -90.000,B 90.000,C 0.000} C_DIS
LIN {X -99.567,Y -25.308,Z -50.088,A -90.000,B 90.000,C 0.000} C_DIS
LIN {X -99.685,Y -25.308,Z -49.757,A -90.000,B 90.000,C 0.000} C_DIS
LIN {X -99.801,Y -25.308,Z -49.384,A -90.000,B 90.000,C 0.000} C_DIS
LIN {X -99.888,Y -25.308,Z -49.073,A -90.000,B 90.000,C 0.000} C_DIS
LIN {X -99.932,Y -25.308,Z -48.890,A -90.000,B 90.000,C 0.000} C_DIS
LIN {X -99.985,Y -25.308,Z -48.654,A -90.000,B 90.000,C 0.000} C_DIS
LIN {X -100.029,Y -25.308,Z -47.948,A -90.000,B 90.000,C 0.000} C_DIS
LIN {X -100.009,Y -25.308,Z -47.517,A -90.000,B 90.000,C 0.000} C_DIS
LIN {X -99.941,Y -25.308,Z -47.156,A -90.000,B 90.000,C 0.000} C_DIS
LIN {X -99.879,Y -25.308,Z -46.881,A -90.000,B 90.000,C 0.000} C_DIS
LIN {X -99.773,Y -25.308,Z -46.626,A -90.000,B 90.000,C 0.000} C_DIS
LIN {X -99.617,Y -25.308,Z -46.301,A -90.000,B 90.000,C 0.000} C_DIS
LIN {X -99.465,Y -25.308,Z -46.064,A -90.000,B 90.000,C 0.000} C_DIS
LIN {X -99.255,Y -25.308,Z -45.807,A -90.000,B 90.000,C 0.000} C_DIS
LIN {X -99.225,Y -25.308,Z -45.767,A -90.000,B 90.000,C 0.000} C_DIS
LIN {X -99.033,Y -25.308,Z -45.560,A -90.000,B 90.000,C 0.000} C_DIS
LIN {X -98.782,Y -25.308,Z -45.353,A -90.000,B 90.000,C 0.000} C_DIS
LIN {X -98.711,Y -25.308,Z -45.288,A -90.000,B 90.000,C 0.000} C_DIS
LIN {X -98.396,Y -25.308,Z -45.052,A -90.000,B 90.000,C 0.000} C_DIS
LIN {X -98.122,Y -25.308,Z -44.888,A -90.000,B 90.000,C 0.000} C_DIS
LIN {X -97.917,Y -25.308,Z -44.785,A -90.000,B 90.000,C 0.000} C_DIS
LIN {X -97.689,Y -25.308,Z -44.662,A -90.000,B 90.000,C 0.000} C_DIS
LIN {X -97.505,Y -25.308,Z -44.587,A -90.000,B 90.000,C 0.000} C_DIS
LIN {X -97.393,Y -25.308,Z -44.542,A -90.000,B 90.000,C 0.000} C_DIS
LIN {X -96.855,Y -25.308,Z -44.397,A -90.000,B 90.000,C 0.000} C_DIS
LIN {X -96.597,Y -25.308,Z -44.330,A -90.000,B 90.000,C 0.000} C_DIS
LIN {X -96.401,Y -25.308,Z -44.285,A -90.000,B 90.000,C 0.000} C_DIS
LIN {X -96.205,Y -25.308,Z -44.244,A -90.000,B 90.000,C 0.000} C_DIS
LIN {X -95.956,Y -25.308,Z -44.207,A -90.000,B 90.000,C 0.000} C_DIS
LIN {X -95.605,Y -25.308,Z -44.185,A -90.000,B 90.000,C 0.000} C_DIS
LIN {X -94.935,Y -25.308,Z -44.189,A -90.000,B 90.000,C 0.000} C_DIS
LIN {X -94.569,Y -25.308,Z -44.194,A -90.000,B 90.000,C 0.000} C_DIS
LIN {X -94.045,Y -25.308,Z -44.209,A -90.000,B 90.000,C 0.000} C_DIS
LIN {X -93.667,Y -25.308,Z -44.229,A -90.000,B 90.000,C 0.000} C_DIS
LIN {X -93.261,Y -25.308,Z -44.277,A -90.000,B 90.000,C 0.000} C_DIS
LIN {X -93.046,Y -25.308,Z -44.308,A -90.000,B 90.000,C 0.000} C_DIS
LIN {X -92.469,Y -25.308,Z -44.415,A -90.000,B 90.000,C 0.000} C_DIS
LIN {X -91.762,Y -25.308,Z -44.582,A -90.000,B 90.000,C 0.000} C_DIS
LIN {X -91.062,Y -25.308,Z -44.766,A -90.000,B 90.000,C 0.000} C_DIS
LIN {X -90.196,Y -25.308,Z -44.999,A -90.000,B 90.000,C 0.000} C_DIS
LIN {X -90.002,Y -25.308,Z -45.066,A -90.000,B 90.000,C 0.000} C_DIS
LIN {X -89.485,Y -25.308,Z -45.248,A -90.000,B 90.000,C 0.000} C_DIS
LIN {X -89.209,Y -25.308,Z -45.348,A -90.000,B 90.000,C 0.000} C_DIS
LIN {X -88.443,Y -25.308,Z -45.634,A -90.000,B 90.000,C 0.000} C_DIS
LIN {X -88.127,Y -25.308,Z -45.760,A -90.000,B 90.000,C 0.000} C_DIS
LIN {X -88.140,Y -25.308,Z -45.698,A -90.000,B 90.000,C 0.000} C_DIS
LIN {X -88.170,Y -25.308,Z -45.463,A -90.000,B 90.000,C 0.000} C_DIS
LIN {X -88.171,Y -25.308,Z -45.321,A -90.000,B 90.000,C 0.000} C_DIS
LIN {X -88.165,Y -25.308,Z -45.112,A -90.000,B 90.000,C 0.000} C_DIS
LIN {X -88.298,Y -25.308,Z -44.625,A -90.000,B 90.000,C 0.000} C_DIS
LIN {X -88.327,Y -25.308,Z -44.390,A -90.000,B 90.000,C 0.000} C_DIS
LIN {X -88.326,Y -25.308,Z -43.906,A -90.000,B 90.000,C 0.000} C_DIS
LIN {X -88.388,Y -25.308,Z -43.535,A -90.000,B 90.000,C 0.000} C_DIS
LIN {X -88.416,Y -25.308,Z -43.319,A -90.000,B 90.000,C 0.000} C_DIS
LIN {X -88.396,Y -25.308,Z -43.083,A -90.000,B 90.000,C 0.000} C_DIS
LIN {X -88.352,Y -25.308,Z -42.659,A -90.000,B 90.000,C 0.000} C_DIS
LIN {X -88.327,Y -25.308,Z -42.258,A -90.000,B 90.000,C 0.000} C_DIS
LIN {X -88.308,Y -25.308,Z -42.034,A -90.000,B 90.000,C 0.000} C_DIS
LIN {X -88.239,Y -25.308,Z -41.808,A -90.000,B 90.000,C 0.000} C_DIS
LIN {X -88.096,Y -25.308,Z -41.369,A -90.000,B 90.000,C 0.000} C_DIS
LIN {X -87.981,Y -25.308,Z -41.162,A -90.000,B 90.000,C 0.000} C_DIS
LIN {X -87.809,Y -25.308,Z -40.965,A -90.000,B 90.000,C 0.000} C_DIS
LIN {X -87.582,Y -25.308,Z -40.493,A -90.000,B 90.000,C 0.000} C_DIS
LIN {X -87.568,Y -25.308,Z -40.468,A -90.000,B 90.000,C 0.000} C_DIS
LIN {X -87.434,Y -25.308,Z -40.260,A -90.000,B 90.000,C 0.000} C_DIS
LIN {X -87.246,Y -25.308,Z -40.057,A -90.000,B 90.000,C 0.000} C_DIS
LIN {X -87.211,Y -25.308,Z -40.028,A -90.000,B 90.000,C 0.000} C_DIS
LIN {X -86.690,Y -25.308,Z -39.638,A -90.000,B 90.000,C 0.000} C_DIS
LIN {X -86.467,Y -25.308,Z -39.411,A -90.000,B 90.000,C 0.000} C_DIS
LIN {X -86.242,Y -25.308,Z -39.241,A -90.000,B 90.000,C 0.000} C_DIS
LIN {X -85.990,Y -25.308,Z -39.114,A -90.000,B 90.000,C 0.000} C_DIS
LIN {X -85.892,Y -25.308,Z -39.066,A -90.000,B 90.000,C 0.000} C_DIS
LIN {X -85.296,Y -25.308,Z -38.691,A -90.000,B 90.000,C 0.000} C_DIS
LIN {X -85.044,Y -25.308,Z -38.564,A -90.000,B 90.000,C 0.000} C_DIS
LIN {X -84.778,Y -25.308,Z -38.485,A -90.000,B 90.000,C 0.000} C_DIS
LIN {X -84.047,Y -25.308,Z -38.289,A -90.000,B 90.000,C 0.000} C_DIS
LIN {X -83.526,Y -25.308,Z -38.128,A -90.000,B 90.000,C 0.000} C_DIS
LIN {X -83.131,Y -25.308,Z -38.010,A -90.000,B 90.000,C 0.000} C_DIS
LIN {X -83.067,Y -25.308,Z -37.995,A -90.000,B 90.000,C 0.000} C_DIS
LIN {X -82.845,Y -25.308,Z -37.970,A -90.000,B 90.000,C 0.000} C_DIS
LIN {X -82.779,Y -25.308,Z -37.965,A -90.000,B 90.000,C 0.000} C_DIS
LIN {X -81.437,Y -25.308,Z -37.927,A -90.000,B 90.000,C 0.000} C_DIS
LIN {X -81.146,Y -25.308,Z -37.912,A -90.000,B 90.000,C 0.000} C_DIS
LIN {X -81.006,Y -25.308,Z -37.915,A -90.000,B 90.000,C 0.000} C_DIS
LIN {X -80.688,Y -25.308,Z -37.942,A -90.000,B 90.000,C 0.000} C_DIS
LIN {X -79.437,Y -25.308,Z -38.131,A -90.000,B 90.000,C 0.000} C_DIS
LIN {X -79.217,Y -25.308,Z -38.160,A -90.000,B 90.000,C 0.000} C_DIS
LIN {X -79.027,Y -25.308,Z -38.190,A -90.000,B 90.000,C 0.000} C_DIS
LIN {X -78.717,Y -25.308,Z -38.266,A -90.000,B 90.000,C 0.000} C_DIS
LIN {X -77.084,Y -25.308,Z -38.699,A -90.000,B 90.000,C 0.000} C_DIS
LIN {X -75.525,Y -25.308,Z -39.179,A -90.000,B 90.000,C 0.000} C_DIS
LIN {X -74.968,Y -25.308,Z -39.330,A -90.000,B 90.000,C 0.000} C_DIS
LIN {X -74.068,Y -25.308,Z -39.571,A -90.000,B 90.000,C 0.000} C_DIS
LIN {X -73.252,Y -25.308,Z -39.794,A -90.000,B 90.000,C 0.000} C_DIS
LIN {X -72.605,Y -25.308,Z -39.967,A -90.000,B 90.000,C 0.000} C_DIS
LIN {X -71.524,Y -25.308,Z -40.304,A -90.000,B 90.000,C 0.000} C_DIS
LIN {X -71.033,Y -25.308,Z -40.454,A -90.000,B 90.000,C 0.000} C_DIS
LIN {X -69.245,Y -25.308,Z -41.122,A -90.000,B 90.000,C 0.000} C_DIS
LIN {X -68.951,Y -25.308,Z -41.245,A -90.000,B 90.000,C 0.000} C_DIS
LIN {X -66.844,Y -25.308,Z -42.183,A -90.000,B 90.000,C 0.000} C_DIS
LIN {X -66.343,Y -25.308,Z -42.413,A -90.000,B 90.000,C 0.000} C_DIS
LIN {X -64.555,Y -25.308,Z -43.247,A -90.000,B 90.000,C 0.000} C_DIS
LIN {X -62.249,Y -25.308,Z -44.259,A -90.000,B 90.000,C 0.000} C_DIS
LIN {X -59.594,Y -25.308,Z -45.270,A -90.000,B 90.000,C 0.000} C_DIS
LIN {X -57.285,Y -25.308,Z -45.957,A -90.000,B 90.000,C 0.000} C_DIS
LIN {X -56.902,Y -25.308,Z -46.076,A -90.000,B 90.000,C 0.000} C_DIS
LIN {X -55.661,Y -25.308,Z -46.358,A -90.000,B 90.000,C 0.000} C_DIS
LIN {X -54.366,Y -25.308,Z -46.676,A -90.000,B 90.000,C 0.000} C_DIS
LIN {X -53.815,Y -25.308,Z -46.770,A -90.000,B 90.000,C 0.000} C_DIS
LIN {X -52.930,Y -25.308,Z -46.942,A -90.000,B 90.000,C 0.000} C_DIS
LIN {X -51.514,Y -25.308,Z -47.276,A -90.000,B 90.000,C 0.000} C_DIS
LIN {X -50.810,Y -25.308,Z -47.424,A -90.000,B 90.000,C 0.000} C_DIS
LIN {X -48.468,Y -25.308,Z -47.907,A -90.000,B 90.000,C 0.000} C_DIS
LIN {X -47.462,Y -25.308,Z -48.083,A -90.000,B 90.000,C 0.000} C_DIS
LIN {X -45.826,Y -25.308,Z -48.396,A -90.000,B 90.000,C 0.000} C_DIS
LIN {X -45.607,Y -25.308,Z -48.440,A -90.000,B 90.000,C 0.000} C_DIS
LIN {X -45.467,Y -25.308,Z -48.471,A -90.000,B 90.000,C 0.000} C_DIS
LIN {X -43.681,Y -25.308,Z -48.812,A -90.000,B 90.000,C 0.000} C_DIS
LIN {X -42.408,Y -25.308,Z -49.069,A -90.000,B 90.000,C 0.000} C_DIS
LIN {X -41.720,Y -25.308,Z -49.198,A -90.000,B 90.000,C 0.000} C_DIS
LIN {X -40.183,Y -25.308,Z -49.503,A -90.000,B 90.000,C 0.000} C_DIS
LIN {X -39.718,Y -25.308,Z -49.597,A -90.000,B 90.000,C 0.000} C_DIS
LIN {X -39.327,Y -25.308,Z -49.684,A -90.000,B 90.000,C 0.000} C_DIS
LIN {X -37.650,Y -25.308,Z -50.042,A -90.000,B 90.000,C 0.000} C_DIS
LIN {X -37.307,Y -25.308,Z -50.119,A -90.000,B 90.000,C 0.000} C_DIS
LIN {X -35.923,Y -25.308,Z -50.445,A -90.000,B 90.000,C 0.000} C_DIS
LIN {X -33.991,Y -25.308,Z -50.936,A -90.000,B 90.000,C 0.000} C_DIS
LIN {X -32.848,Y -25.308,Z -51.214,A -90.000,B 90.000,C 0.000} C_DIS
LIN {X -30.149,Y -25.308,Z -51.936,A -90.000,B 90.000,C 0.000} C_DIS
LIN {X -30.024,Y -25.308,Z -51.967,A -90.000,B 90.000,C 0.000} C_DIS
LIN {X -29.595,Y -25.308,Z -52.082,A -90.000,B 90.000,C 0.000} C_DIS
LIN {X -27.356,Y -25.308,Z -52.714,A -90.000,B 90.000,C 0.000} C_DIS
LIN {X -25.439,Y -25.308,Z -53.220,A -90.000,B 90.000,C 0.000} C_DIS
LIN {X -25.125,Y -25.308,Z -53.304,A -90.000,B 90.000,C 0.000} C_DIS
LIN {X -23.354,Y -25.308,Z -53.723,A -90.000,B 90.000,C 0.000} C_DIS
LIN {X -22.934,Y -25.308,Z -53.808,A -90.000,B 90.000,C 0.000} C_DIS
LIN {X -22.075,Y -25.308,Z -53.953,A -90.000,B 90.000,C 0.000} C_DIS
LIN {X -21.560,Y -25.308,Z -54.003,A -90.000,B 90.000,C 0.000} C_DIS
LIN {X -21.080,Y -25.308,Z -54.029,A -90.000,B 90.000,C 0.000} C_DIS
LIN {X -20.950,Y -25.308,Z -54.023,A -90.000,B 90.000,C 0.000} C_DIS
LIN {X -20.373,Y -25.308,Z -53.970,A -90.000,B 90.000,C 0.000} C_DIS
LIN {X -19.767,Y -25.308,Z -53.818,A -90.000,B 90.000,C 0.000} C_DIS
LIN {X -19.395,Y -25.308,Z -53.744,A -90.000,B 90.000,C 0.000} C_DIS
LIN {X -18.980,Y -25.308,Z -53.604,A -90.000,B 90.000,C 0.000} C_DIS
LIN {X -18.445,Y -25.308,Z -53.441,A -90.000,B 90.000,C 0.000} C_DIS
LIN {X -17.331,Y -25.308,Z -53.031,A -90.000,B 90.000,C 0.000} C_DIS
LIN {X -17.166,Y -25.308,Z -52.972,A -90.000,B 90.000,C 0.000} C_DIS
LIN {X -16.007,Y -25.308,Z -52.584,A -90.000,B 90.000,C 0.000} C_DIS
LIN {X -15.815,Y -25.308,Z -52.521,A -90.000,B 90.000,C 0.000} C_DIS
LIN {X -15.479,Y -25.308,Z -52.417,A -90.000,B 90.000,C 0.000} C_DIS
LIN {X -15.354,Y -25.308,Z -52.381,A -90.000,B 90.000,C 0.000} C_DIS
LIN {X -15.213,Y -25.308,Z -52.354,A -90.000,B 90.000,C 0.000} C_DIS
LIN {X -14.285,Y -25.308,Z -52.147,A -90.000,B 90.000,C 0.000} C_DIS
LIN {X -13.786,Y -25.308,Z -52.049,A -90.000,B 90.000,C 0.000} C_DIS
LIN {X -12.768,Y -25.308,Z -51.887,A -90.000,B 90.000,C 0.000} C_DIS
LIN {X -12.690,Y -25.308,Z -51.876,A -90.000,B 90.000,C 0.000} C_DIS
LIN {X -12.608,Y -25.308,Z -51.869,A -90.000,B 90.000,C 0.000} C_DIS
LIN {X -11.702,Y -25.308,Z -51.770,A -90.000,B 90.000,C 0.000} C_DIS
LIN {X -10.505,Y -25.308,Z -51.700,A -90.000,B 90.000,C 0.000} C_DIS
LIN {X -10.266,Y -25.308,Z -51.682,A -90.000,B 90.000,C 0.000} C_DIS
LIN {X -10.076,Y -25.308,Z -51.675,A -90.000,B 90.000,C 0.000} C_DIS
LIN {X -9.931,Y -25.308,Z -51.667,A -90.000,B 90.000,C 0.000} C_DIS
LIN {X -9.073,Y -25.308,Z -51.647,A -90.000,B 90.000,C 0.000} C_DIS
LIN {X -9.016,Y -25.308,Z -51.649,A -90.000,B 90.000,C 0.000} C_DIS
LIN {X -8.312,Y -25.308,Z -51.647,A -90.000,B 90.000,C 0.000} C_DIS
LIN {X -8.081,Y -25.308,Z -51.651,A -90.000,B 90.000,C 0.000} C_DIS
LIN {X -7.869,Y -25.308,Z -51.658,A -90.000,B 90.000,C 0.000} C_DIS
LIN {X -6.073,Y -25.308,Z -51.700,A -90.000,B 90.000,C 0.000} C_DIS
LIN {X -5.633,Y -25.308,Z -51.717,A -90.000,B 90.000,C 0.000} C_DIS
LIN {X -4.137,Y -25.308,Z -51.802,A -90.000,B 90.000,C 0.000} C_DIS
LIN {X -3.604,Y -25.308,Z -51.827,A -90.000,B 90.000,C 0.000} C_DIS
LIN {X -3.288,Y -25.308,Z -51.854,A -90.000,B 90.000,C 0.000} C_DIS
LIN {X -2.820,Y -25.308,Z -51.876,A -90.000,B 90.000,C 0.000} C_DIS
LIN {X -0.713,Y -25.308,Z -52.021,A -90.000,B 90.000,C 0.000} C_DIS
LIN {X -0.279,Y -25.308,Z -52.062,A -90.000,B 90.000,C 0.000} C_DIS
LIN {X 0.570,Y -25.308,Z -52.079,A -90.000,B 90.000,C 0.000} C_DIS
LIN {X 1.129,Y -25.308,Z -52.099,A -90.000,B 90.000,C 0.000} C_DIS
LIN {X 1.237,Y -25.308,Z -52.092,A -90.000,B 90.000,C 0.000} C_DIS
LIN {X 2.358,Y -25.308,Z -52.052,A -90.000,B 90.000,C 0.000} C_DIS
LIN {X 2.428,Y -25.308,Z -52.048,A -90.000,B 90.000,C 0.000} C_DIS
LIN {X 3.349,Y -25.308,Z -51.974,A -90.000,B 90.000,C 0.000} C_DIS
LIN {X 3.681,Y -25.308,Z -51.952,A -90.000,B 90.000,C 0.000} C_DIS
LIN {X 4.621,Y -25.308,Z -51.915,A -90.000,B 90.000,C 0.000} C_DIS
LIN {X 4.856,Y -25.308,Z -51.911,A -90.000,B 90.000,C 0.000} C_DIS
LIN {X 4.978,Y -25.308,Z -51.917,A -90.000,B 90.000,C 0.000} C_DIS
LIN {X 5.962,Y -25.308,Z -51.927,A -90.000,B 90.000,C 0.000} C_DIS
LIN {X 6.501,Y -25.308,Z -51.949,A -90.000,B 90.000,C 0.000} C_DIS
LIN {X 8.603,Y -25.308,Z -52.069,A -90.000,B 90.000,C 0.000} C_DIS
LIN {X 9.580,Y -25.308,Z -52.165,A -90.000,B 90.000,C 0.000} C_DIS
LIN {X 9.978,Y -25.308,Z -52.223,A -90.000,B 90.000,C 0.000} C_DIS
LIN {X 10.622,Y -25.308,Z -52.333,A -90.000,B 90.000,C 0.000} C_DIS
LIN {X 10.913,Y -25.308,Z -52.396,A -90.000,B 90.000,C 0.000} C_DIS
LIN {X 12.735,Y -25.308,Z -52.821,A -90.000,B 90.000,C 0.000} C_DIS
LIN {X 13.725,Y -25.308,Z -53.010,A -90.000,B 90.000,C 0.000} C_DIS
LIN {X 14.128,Y -25.308,Z -53.090,A -90.000,B 90.000,C 0.000} C_DIS
LIN {X 15.179,Y -25.308,Z -53.273,A -90.000,B 90.000,C 0.000} C_DIS
LIN {X 15.517,Y -25.308,Z -53.325,A -90.000,B 90.000,C 0.000} C_DIS
LIN {X 15.784,Y -25.308,Z -52.633,A -90.000,B 90.000,C 0.000} C_DIS
LIN {X 15.956,Y -25.308,Z -52.327,A -90.000,B 90.000,C 0.000} C_DIS
LIN {X 16.527,Y -25.308,Z -51.552,A -90.000,B 90.000,C 0.000} C_DIS
LIN {X 16.807,Y -25.308,Z -51.184,A -90.000,B 90.000,C 0.000} C_DIS
LIN {X 17.459,Y -25.308,Z -50.542,A -90.000,B 90.000,C 0.000} C_DIS
LIN {X 17.972,Y -25.308,Z -50.082,A -90.000,B 90.000,C 0.000} C_DIS
LIN {X 18.022,Y -25.308,Z -50.043,A -90.000,B 90.000,C 0.000} C_DIS
